  MoveL 6563 to (20.68, -72.48, -149.47) mm, rotated rx 105.8 ry 33.04 rz 34.05 deg; joints [-5.945, -30.892, 104.266, 145.331, 85.223, 18.714, -475]
  MoveL 6564 to (20.48, -73.16, -150.23) mm, rotated rx 105.8 ry 33.04 rz 34.05 deg; joints [-5.975, -30.911, 104.238, 145.3, 85.188, 18.748, -475]
  MoveL 6565 to (19.98, -73.73, -151.16) mm, rotated rx 105.8 ry 33.04 rz 34.05 deg; joints [-6.01, -30.911, 104.183, 145.262, 85.15, 18.787, -475]
  MoveL 6566 to (18.11, -74.59, -153.52) mm, rotated rx 105.8 ry 33.04 rz 34.05 deg; joints [-6.101, -30.851, 103.995, 145.167, 85.06, 18.882, -475]
  MoveL 6567 to (15.72, -74.84, -155.88) mm, rotated rx 105.8 ry 33.04 rz 34.05 deg; joints [-6.192, -30.738, 103.766, 145.073, 84.979, 18.97, -475]
  MoveL 6568 to (13.46, -74.3, -157.57) mm, rotated rx 105.8 ry 33.04 rz 34.05 deg; joints [-6.256, -30.597, 103.559, 145.006, 84.936, 19.024, -475]
  MoveL 6569 to (12.38, -73.73, -158.16) mm, rotated rx 105.8 ry 33.04 rz 34.05 deg; joints [-6.279, -30.516, 103.464, 144.984, 84.929, 19.037, -475]
  MoveL 6570 to (11.34, -72.97, -158.58) mm, rotated rx 105.8 ry 33.04 rz 34.05 deg; joints [-6.295, -30.429, 103.375, 144.968, 84.93, 19.042, -475]
  MoveL 6571 to (9.34, -70.84, -158.92) mm, rotated rx 105.8 ry 33.04 rz 34.05 deg; joints [-6.308, -30.233, 103.215, 144.957, 84.961, 19.025, -475]
  MoveL 6572 to (6.8, -67.51, -158.92) mm, rotated rx 105.8 ry 33.04 rz 34.05 deg; joints [-6.309, -29.957, 103.017, 144.96, 85.025, 18.98, -475]
  MoveL 6573 to (6.45, -67.09, -158.94) mm, rotated rx 105.8 ry 33.04 rz 34.05 deg; joints [-6.309, -29.921, 102.99, 144.96, 85.033, 18.975, -475]
  MoveL 6574 to (6.11, -66.68, -158.98) mm, rotated rx 105.8 ry 33.04 rz 34.05 deg; joints [-6.311, -29.886, 102.962, 144.959, 85.039, 18.971, -475]
  MoveL 6575 to (5.76, -66.29, -159.04) mm, rotated rx 105.8 ry 33.04 rz 34.05 deg; joints [-6.313, -29.85, 102.934, 144.957, 85.045, 18.968, -475]
  MoveL 6576 to (5.4, -65.92, -159.12) mm, rotated rx 105.8 ry 33.04 rz 34.05 deg; joints [-6.317, -29.815, 102.904, 144.954, 85.05, 18.965, -475]
  MoveL 6577 to (5.05, -65.55, -159.2) mm, rotated rx 105.8 ry 33.04 rz 34.05 deg; joints [-6.32, -29.781, 102.876, 144.951, 85.055, 18.963, -475]
  MoveL 6578 to (4.73, -65.18, -159.24) mm, rotated rx 105.8 ry 33.04 rz 34.05 deg; joints [-6.321, -29.749, 102.85, 144.95, 85.061, 18.959, -475]
  MoveL 6579 to (4.43, -64.8, -159.25) mm, rotated rx 105.8 ry 33.04 rz 34.05 deg; joints [-6.322, -29.717, 102.826, 144.95, 85.068, 18.955, -475]
  MoveL 6580 to (4.11, -64.39, -159.25) mm, rotated rx 105.8 ry 33.04 rz 34.05 deg; joints [-6.322, -29.683, 102.801, 144.95, 85.076, 18.949, -475]
  MoveL 6581 to (3.72, -63.9, -159.29) mm, rotated rx 105.8 ry 33.04 rz 34.05 deg; joints [-6.323, -29.641, 102.77, 144.949, 85.084, 18.944, -475]
  MoveL 6582 to (3.27, -63.39, -159.35) mm, rotated rx 105.8 ry 33.04 rz 34.05 deg; joints [-6.326, -29.596, 102.734, 144.947, 85.092, 18.939, -475]
  MoveL 6583 to (2.88, -62.94, -159.37) mm, rotated rx 105.8 ry 33.04 rz 34.05 deg; joints [-6.326, -29.556, 102.702, 144.947, 85.099, 18.934, -475]
  MoveL 6584 to (2.49, -62.55, -159.38) mm, rotated rx 105.8 ry 33.04 rz 34.05 deg; joints [-6.327, -29.518, 102.67, 144.947, 85.103, 18.932, -475]
  MoveL 6585 to (2.06, -62.19, -159.38) mm, rotated rx 105.8 ry 33.04 rz 34.05 deg; joints [-6.327, -29.481, 102.634, 144.947, 85.104, 18.931, -475]
  MoveL 6586 to (1.55, -61.92, -159.38) mm, rotated rx 105.8 ry 33.04 rz 34.05 deg; joints [-6.326, -29.443, 102.589, 144.947, 85.099, 18.935, -475]
  MoveL 6587 to (0.98, -61.7, -159.38) mm, rotated rx 105.8 ry 33.04 rz 34.05 deg; joints [-6.326, -29.404, 102.539, 144.947, 85.089, 18.941, -475]
  MoveL 6588 to (2.28, -62.59, -160.34) mm, rotated rx 105.8 ry 33.04 rz 34.05 deg; joints [-6.364, -29.51, 102.648, 144.91, 85.098, 18.948, -475]
  MoveL 6589 to (1.05, -62.41, -160.76) mm, rotated rx 105.8 ry 33.04 rz 34.05 deg; joints [-6.379, -29.438, 102.533, 144.893, 85.066, 18.977, -475]
  MoveL 6590 to (-0.34, -62.11, -161.09) mm, rotated rx 105.8 ry 33.04 rz 34.05 deg; joints [-6.391, -29.353, 102.406, 144.879, 85.033, 19.004, -475]
  MoveL 6591 to (-1.89, -61.69, -161.34) mm, rotated rx 105.8 ry 33.04 rz 34.05 deg; joints [-6.4, -29.255, 102.265, 144.869, 84.999, 19.031, -475]
  MoveL 6592 to (-3.92, -61.03, -161.45) mm, rotated rx 105.8 ry 33.04 rz 34.05 deg; joints [-6.402, -29.121, 102.081, 144.863, 84.959, 19.06, -475]
  MoveL 6593 to (-5.95, -60.38, -161.68) mm, rotated rx 105.8 ry 33.04 rz 34.05 deg; joints [-6.41, -28.988, 101.897, 144.854, 84.918, 19.091, -475]
  MoveL 6594 to (-7.97, -59.71, -161.79) mm, rotated rx 105.8 ry 33.04 rz 34.05 deg; joints [-6.413, -28.854, 101.713, 144.848, 84.878, 19.121, -475]
  MoveL 6595 to (-10, -59.04, -161.91) mm, rotated rx 105.8 ry 33.04 rz 34.05 deg; joints [-6.416, -28.72, 101.529, 144.843, 84.838, 19.151, -475]
  MoveL 6596 to (-12.02, -58.38, -162.14) mm, rotated rx 105.8 ry 33.04 rz 34.05 deg; joints [-6.424, -28.587, 101.344, 144.832, 84.797, 19.182, -475]
  MoveL 6597 to (-14.05, -57.7, -162.27) mm, rotated rx 105.8 ry 33.04 rz 34.05 deg; joints [-6.427, -28.453, 101.16, 144.827, 84.756, 19.212, -475]
  MoveL 6598 to (-16.07, -57.02, -162.38) mm, rotated rx 105.8 ry 33.04 rz 34.05 deg; joints [-6.43, -28.318, 100.975, 144.821, 84.716, 19.242, -475]
  MoveL 6599 to (-18.4, -56.24, -162.54) mm, rotated rx 105.8 ry 33.04 rz 34.05 deg; joints [-6.434, -28.164, 100.761, 144.813, 84.668, 19.277, -475]
  MoveL 6600 to (-20.39, -55.57, -162.74) mm, rotated rx 105.8 ry 33.04 rz 34.05 deg; joints [-6.44, -28.031, 100.579, 144.805, 84.628, 19.308, -475]
  MoveL 6601 to (-22.58, -54.83, -162.94) mm, rotated rx 105.8 ry 33.04 rz 34.05 deg; joints [-6.446, -27.885, 100.378, 144.796, 84.584, 19.342, -475]
  MoveL 6602 to (-24.71, -54.09, -163.19) mm, rotated rx 105.8 ry 33.04 rz 34.05 deg; joints [-6.454, -27.743, 100.18, 144.785, 84.541, 19.375, -475]
  MoveL 6603 to (-26.73, -53.4, -163.31) mm, rotated rx 105.8 ry 33.04 rz 34.05 deg; joints [-6.458, -27.608, 99.994, 144.779, 84.5, 19.406, -475]
  MoveL 6604 to (-28.75, -52.71, -163.31) mm, rotated rx 105.8 ry 33.04 rz 34.05 deg; joints [-6.456, -27.473, 99.808, 144.777, 84.457, 19.435, -475]
  MoveL 6605 to (-30.74, -52.02, -163.39) mm, rotated rx 105.8 ry 33.04 rz 34.05 deg; joints [-6.458, -27.34, 99.624, 144.773, 84.416, 19.465, -475]
  MoveL 6606 to (-32.68, -51.33, -163.6) mm, rotated rx 105.8 ry 33.04 rz 34.05 deg; joints [-6.465, -27.209, 99.444, 144.764, 84.377, 19.495, -475]
  MoveL 6607 to (-34.84, -50.54, -163.95) mm, rotated rx 105.8 ry 33.04 rz 34.05 deg; joints [-6.476, -27.062, 99.243, 144.749, 84.335, 19.53, -475]
  MoveL 6608 to (-36.54, -49.92, -164.16) mm, rotated rx 105.8 ry 33.04 rz 34.05 deg; joints [-6.483, -26.947, 99.085, 144.74, 84.301, 19.556, -475]
  MoveL 6609 to (-38.84, -49.05, -164.46) mm, rotated rx 105.8 ry 33.04 rz 34.05 deg; joints [-6.493, -26.79, 98.871, 144.727, 84.256, 19.592, -475]
  MoveL 6610 to (-40.92, -48.31, -164.57) mm, rotated rx 105.8 ry 33.04 rz 34.05 deg; joints [-6.496, -26.649, 98.676, 144.721, 84.213, 19.624, -475]
  MoveL 6611 to (-42.93, -47.62, -164.58) mm, rotated rx 105.8 ry 33.04 rz 34.05 deg; joints [-6.495, -26.515, 98.488, 144.719, 84.169, 19.655, -475]
  MoveL 6612 to (-43.47, -46.91, -165.37) mm, rotated rx 105.8 ry 33.04 rz 34.05 deg; joints [-6.525, -26.456, 98.44, 144.69, 84.183, 19.656, -475]
  MoveL 6613 to (-43.03, -46.88, -165.76) mm, rotated rx 105.8 ry 33.04 rz 34.05 deg; joints [-6.54, -26.477, 98.482, 144.677, 84.203, 19.648, -475]
  MoveL 6614 to (-42.89, -46.88, -166) mm, rotated rx 105.8 ry 33.04 rz 34.05 deg; joints [-6.55, -26.484, 98.495, 144.668, 84.209, 19.647, -475]
  MoveL 6615 to (-43.03, -46.91, -166.13) mm, rotated rx 105.8 ry 33.04 rz 34.05 deg; joints [-6.554, -26.479, 98.481, 144.663, 84.203, 19.653, -475]
  MoveL 6616 to (-43.41, -47, -166.15) mm, rotated rx 105.8 ry 33.04 rz 34.05 deg; joints [-6.554, -26.462, 98.442, 144.661, 84.185, 19.666, -475]
  MoveL 6617 to (-43.87, -47.11, -166.16) mm, rotated rx 105.8 ry 33.04 rz 34.05 deg; joints [-6.554, -26.443, 98.397, 144.66, 84.164, 19.681, -475]
  MoveL 6618 to (-45.38, -47.52, -166.16) mm, rotated rx 105.8 ry 33.04 rz 34.05 deg; joints [-6.552, -26.381, 98.246, 144.657, 84.091, 19.732, -475]
  MoveL 6619 to (-45.92, -47.65, -166.18) mm, rotated rx 105.8 ry 33.04 rz 34.05 deg; joints [-6.552, -26.358, 98.192, 144.655, 84.065, 19.75, -475]
  MoveL 6620 to (-46.46, -47.77, -166.22) mm, rotated rx 105.8 ry 33.04 rz 34.05 deg; joints [-6.553, -26.334, 98.138, 144.652, 84.041, 19.768, -475]
  MoveL 6621 to (-47.03, -47.86, -166.31) mm, rotated rx 105.8 ry 33.04 rz 34.05 deg; joints [-6.556, -26.309, 98.082, 144.648, 84.017, 19.786, -475]
  MoveL 6622 to (-47.57, -47.97, -166.37) mm, rotated rx 105.8 ry 33.04 rz 34.05 deg; joints [-6.557, -26.284, 98.028, 144.644, 83.992, 19.804, -475]
  MoveL 6623 to (-48.09, -48.09, -166.39) mm, rotated rx 105.8 ry 33.04 rz 34.05 deg; joints [-6.558, -26.262, 97.976, 144.642, 83.968, 19.821, -475]
  MoveL 6624 to (-48.57, -48.2, -166.41) mm, rotated rx 105.8 ry 33.04 rz 34.05 deg; joints [-6.558, -26.242, 97.928, 144.64, 83.946, 19.838, -475]
  MoveL 6625 to (-49.02, -48.29, -166.45) mm, rotated rx 105.8 ry 33.04 rz 34.05 deg; joints [-6.559, -26.222, 97.883, 144.638, 83.926, 19.852, -475]
  MoveL 6626 to (-49.45, -48.38, -166.49) mm, rotated rx 105.8 ry 33.04 rz 34.05 deg; joints [-6.56, -26.202, 97.839, 144.635, 83.906, 19.867, -475]
  MoveL 6627 to (-49.94, -48.5, -166.51) mm, rotated rx 105.8 ry 33.04 rz 34.05 deg; joints [-6.56, -26.182, 97.791, 144.634, 83.883, 19.883, -475]
  MoveL 6628 to (-50.51, -48.63, -166.53) mm, rotated rx 105.8 ry 33.04 rz 34.05 deg; joints [-6.56, -26.158, 97.734, 144.632, 83.857, 19.902, -475]
  MoveL 6629 to (-51.19, -48.77, -166.58) mm, rotated rx 105.8 ry 33.04 rz 34.05 deg; joints [-6.561, -26.127, 97.665, 144.628, 83.825, 19.925, -475]
  MoveL 6630 to (-51.78, -48.91, -166.61) mm, rotated rx 105.8 ry 33.04 rz 34.05 deg; joints [-6.561, -26.102, 97.606, 144.626, 83.798, 19.944, -475]
  MoveL 6631 to (-53.82, -49.45, -166.61) mm, rotated rx 105.8 ry 33.04 rz 34.05 deg; joints [-6.559, -26.017, 97.401, 144.62, 83.7, 20.014, -475]
  MoveL 6632 to (-56.69, -49.93, -166.94) mm, rotated rx 105.8 ry 33.04 rz 34.05 deg; joints [-6.568, -25.885, 97.113, 144.602, 83.575, 20.106, -475]
  MoveL 6633 to (-57.98, -49.9, -167.35) mm, rotated rx 105.8 ry 33.04 rz 34.05 deg; joints [-6.582, -25.815, 96.985, 144.584, 83.53, 20.144, -475]
  MoveL 6634 to (-59.18, -49.7, -167.93) mm, rotated rx 105.8 ry 33.04 rz 34.05 deg; joints [-6.602, -25.742, 96.867, 144.561, 83.497, 20.176, -475]
  MoveL 6635 to (-61.29, -48.77, -169.58) mm, rotated rx 105.8 ry 33.04 rz 34.05 deg; joints [-6.663, -25.59, 96.664, 144.498, 83.466, 20.222, -475]
  MoveL 6636 to (-63.02, -47.13, -171.89) mm, rotated rx 105.8 ry 33.04 rz 34.05 deg; joints [-6.749, -25.429, 96.502, 144.414, 83.482, 20.246, -475]
  MoveL 6637 to (-63.97, -45.34, -174.19) mm, rotated rx 105.8 ry 33.04 rz 34.05 deg; joints [-6.837, -25.302, 96.418, 144.331, 83.533, 20.244, -475]
  MoveL 6638 to (-64, -44.59, -175.1) mm, rotated rx 105.8 ry 33.04 rz 34.05 deg; joints [-6.872, -25.269, 96.418, 144.3, 83.567, 20.233, -475]
  MoveL 6639 to (-63.75, -43.94, -175.84) mm, rotated rx 105.8 ry 33.04 rz 34.05 deg; joints [-6.9, -25.255, 96.447, 144.274, 83.608, 20.215, -475]
  MoveL 6640 to (-63.51, -43.65, -176.15) mm, rotated rx 105.8 ry 33.04 rz 34.05 deg; joints [-6.913, -25.255, 96.472, 144.264, 83.63, 20.204, -475]
  MoveL 6641 to (-63.2, -43.39, -176.42) mm, rotated rx 105.8 ry 33.04 rz 34.05 deg; joints [-6.923, -25.26, 96.505, 144.255, 83.654, 20.191, -475]
  MoveL 6642 to (-62.36, -42.93, -176.83) mm, rotated rx 105.8 ry 33.04 rz 34.05 deg; joints [-6.94, -25.286, 96.591, 144.243, 83.707, 20.16, -475]
  MoveL 6643 to (-61.22, -42.58, -177.08) mm, rotated rx 105.8 ry 33.04 rz 34.05 deg; joints [-6.952, -25.33, 96.705, 144.236, 83.765, 20.122, -475]
  MoveL 6644 to (-59.79, -42.31, -177.16) mm, rotated rx 105.8 ry 33.04 rz 34.05 deg; joints [-6.957, -25.395, 96.848, 144.236, 83.83, 20.077, -475]
  MoveL 6645 to (-56.16, -41.83, -177.16) mm, rotated rx 105.8 ry 33.04 rz 34.05 deg; joints [-6.962, -25.566, 97.211, 144.243, 83.986, 19.966, -475]
  MoveL 6646 to (-55.7, -41.77, -177.14) mm, rotated rx 105.8 ry 33.04 rz 34.05 deg; joints [-6.962, -25.588, 97.256, 144.244, 84.005, 19.952, -475]
  MoveL 6647 to (-55.29, -41.74, -177.12) mm, rotated rx 105.8 ry 33.04 rz 34.05 deg; joints [-6.962, -25.608, 97.297, 144.246, 84.022, 19.94, -475]
  MoveL 6648 to (-54.82, -41.69, -177.1) mm, rotated rx 105.8 ry 33.04 rz 34.05 deg; joints [-6.962, -25.631, 97.344, 144.247, 84.041, 19.926, -475]
  MoveL 6649 to (-51.19, -41.2, -177.1) mm, rotated rx 105.8 ry 33.04 rz 34.05 deg; joints [-6.967, -25.801, 97.704, 144.254, 84.197, 19.815, -475]
  MoveL 6650 to (-50.65, -41.15, -177.08) mm, rotated rx 105.8 ry 33.04 rz 34.05 deg; joints [-6.967, -25.828, 97.758, 144.255, 84.218, 19.8, -475]
  MoveL 6651 to (-50.1, -41.13, -177.04) mm, rotated rx 105.8 ry 33.04 rz 34.05 deg; joints [-6.966, -25.855, 97.811, 144.257, 84.239, 19.784, -475]
  MoveL 6652 to (-49.62, -41.16, -177) mm, rotated rx 105.8 ry 33.04 rz 34.05 deg; joints [-6.965, -25.882, 97.859, 144.26, 84.256, 19.772, -475]
  MoveL 6653 to (-49.24, -41.22, -176.94) mm, rotated rx 105.8 ry 33.04 rz 34.05 deg; joints [-6.963, -25.905, 97.895, 144.262, 84.267, 19.763, -475]
  MoveL 6654 to (-49.06, -41.28, -176.77) mm, rotated rx 105.8 ry 33.04 rz 34.05 deg; joints [-6.957, -25.917, 97.913, 144.269, 84.27, 19.758, -475]
  MoveL 6655 to (-49.05, -41.32, -176.44) mm, rotated rx 105.8 ry 33.04 rz 34.05 deg; joints [-6.945, -25.919, 97.915, 144.281, 84.268, 19.755, -475]
  MoveL 6656 to (-49.2, -41.32, -175.93) mm, rotated rx 105.8 ry 33.04 rz 34.05 deg; joints [-6.925, -25.912, 97.901, 144.3, 84.26, 19.754, -475]
  MoveL 6657 to (-48.89, -42.09, -174.47) mm, rotated rx 105.8 ry 33.04 rz 34.05 deg; joints [-6.869, -25.962, 97.929, 144.353, 84.232, 19.753, -475]
  MoveL 6658 to (-45.07, -43.97, -174.47) mm, rotated rx 105.8 ry 33.04 rz 34.05 deg; joints [-6.872, -26.242, 98.284, 144.354, 84.293, 19.71, -475]
  MoveL 6659 to (-43.24, -44.88, -174.42) mm, rotated rx 105.8 ry 33.04 rz 34.05 deg; joints [-6.872, -26.376, 98.453, 144.357, 84.321, 19.689, -475]
  MoveL 6660 to (-41.47, -45.76, -174.33) mm, rotated rx 105.8 ry 33.04 rz 34.05 deg; joints [-6.87, -26.506, 98.617, 144.361, 84.348, 19.669, -475]
  MoveL 6661 to (-39.66, -46.65, -174.25) mm, rotated rx 105.8 ry 33.04 rz 34.05 deg; joints [-6.868, -26.639, 98.784, 144.364, 84.375, 19.649, -475]
  MoveL 6662 to (-37.89, -47.52, -174.15) mm, rotated rx 105.8 ry 33.04 rz 34.05 deg; joints [-6.866, -26.769, 98.946, 144.369, 84.401, 19.629, -475]
  MoveL 6663 to (-36.03, -48.47, -174.11) mm, rotated rx 105.8 ry 33.04 rz 34.05 deg; joints [-6.866, -26.907, 99.117, 144.371, 84.428, 19.61, -475]
  MoveL 6664 to (-34.1, -49.54, -174.07) mm, rotated rx 105.8 ry 33.04 rz 34.05 deg; joints [-6.866, -27.053, 99.292, 144.372, 84.452, 19.593, -475]
  MoveL 6665 to (-31.82, -50.56, -173.91) mm, rotated rx 105.8 ry 33.04 rz 34.05 deg; joints [-6.861, -27.215, 99.502, 144.379, 84.489, 19.564, -475]
  MoveL 6666 to (-29.81, -51.55, -173.66) mm, rotated rx 105.8 ry 33.04 rz 34.05 deg; joints [-6.853, -27.363, 99.686, 144.389, 84.518, 19.54, -475]
  MoveL 6667 to (-27.84, -52.52, -173.53) mm, rotated rx 105.8 ry 33.04 rz 34.05 deg; joints [-6.85, -27.507, 99.866, 144.394, 84.546, 19.519, -475]
  MoveL 6668 to (-25.92, -53.46, -173.29) mm, rotated rx 105.8 ry 33.04 rz 34.05 deg; joints [-6.842, -27.647, 100.04, 144.404, 84.573, 19.497, -475]
  MoveL 6669 to (-24, -54.39, -173.17) mm, rotated rx 105.8 ry 33.04 rz 34.05 deg; joints [-6.839, -27.787, 100.214, 144.409, 84.6, 19.476, -475]
  MoveL 6670 to (-22.08, -55.33, -173.05) mm, rotated rx 105.8 ry 33.04 rz 34.05 deg; joints [-6.836, -27.927, 100.388, 144.414, 84.626, 19.456, -475]
  MoveL 6671 to (-20.16, -56.25, -172.81) mm, rotated rx 105.8 ry 33.04 rz 34.05 deg; joints [-6.828, -28.067, 100.562, 144.423, 84.653, 19.434, -475]
  MoveL 6672 to (-18.24, -57.18, -172.69) mm, rotated rx 105.8 ry 33.04 rz 34.05 deg; joints [-6.825, -28.207, 100.736, 144.428, 84.68, 19.413, -475]
  MoveL 6673 to (-16.32, -58.1, -172.57) mm, rotated rx 105.8 ry 33.04 rz 34.05 deg; joints [-6.822, -28.347, 100.909, 144.432, 84.707, 19.393, -475]
  MoveL 6674 to (-14.39, -59.03, -172.45) mm, rotated rx 105.8 ry 33.04 rz 34.05 deg; joints [-6.819, -28.486, 101.081, 144.437, 84.733, 19.373, -475]
  MoveL 6675 to (-12.46, -59.93, -172.22) mm, rotated rx 105.8 ry 33.04 rz 34.05 deg; joints [-6.812, -28.626, 101.255, 144.446, 84.76, 19.351, -475]
  MoveL 6676 to (-10.53, -60.85, -172.11) mm, rotated rx 105.8 ry 33.04 rz 34.05 deg; joints [-6.809, -28.765, 101.428, 144.451, 84.786, 19.331, -475]
  MoveL 6677 to (-8.9, -61.58, -171.86) mm, rotated rx 105.8 ry 33.04 rz 34.05 deg; joints [-6.801, -28.882, 101.574, 144.46, 84.809, 19.312, -475]
  MoveL 6678 to (-7.39, -62.24, -171.54) mm, rotated rx 105.8 ry 33.04 rz 34.05 deg; joints [-6.789, -28.989, 101.711, 144.473, 84.831, 19.292, -475]
  MoveL 6679 to (-5.94, -62.84, -171.12) mm, rotated rx 105.8 ry 33.04 rz 34.05 deg; joints [-6.774, -29.09, 101.843, 144.489, 84.853, 19.271, -475]
  MoveL 6680 to (-7.04, -61.5, -170.16) mm, rotated rx 105.8 ry 33.04 rz 34.05 deg; joints [-6.737, -28.976, 101.756, 144.527, 84.87, 19.245, -475]
  MoveL 6681 to (-6.5, -61.82, -170.04) mm, rotated rx 105.8 ry 33.04 rz 34.05 deg; joints [-6.733, -29.018, 101.805, 144.532, 84.874, 19.24, -475]
  MoveL 6682 to (-6.03, -62.17, -169.95) mm, rotated rx 105.8 ry 33.04 rz 34.05 deg; joints [-6.729, -29.057, 101.845, 144.535, 84.874, 19.239, -475]
  MoveL 6683 to (-5.66, -62.57, -169.92) mm, rotated rx 105.8 ry 33.04 rz 34.05 deg; joints [-6.728, -29.093, 101.875, 144.536, 84.869, 19.242, -475]
  MoveL 6684 to (-5.35, -63, -169.9) mm, rotated rx 105.8 ry 33.04 rz 34.05 deg; joints [-6.728, -29.128, 101.9, 144.536, 84.861, 19.248, -475]
  MoveL 6685 to (-3.48, -66.17, -169.89) mm, rotated rx 105.8 ry 33.04 rz 34.05 deg; joints [-6.726, -29.361, 102.039, 144.532, 84.784, 19.302, -475]
  MoveL 6686 to (-3.24, -66.57, -169.88) mm, rotated rx 105.8 ry 33.04 rz 34.05 deg; joints [-6.726, -29.391, 102.057, 144.532, 84.775, 19.309, -475]
  MoveL 6687 to (-3.02, -66.92, -169.85) mm, rotated rx 105.8 ry 33.04 rz 34.05 deg; joints [-6.725, -29.418, 102.075, 144.533, 84.766, 19.314, -475]
  MoveL 6688 to (-2.77, -67.33, -169.84) mm, rotated rx 105.8 ry 33.04 rz 34.05 deg; joints [-6.724, -29.449, 102.093, 144.532, 84.756, 19.321, -475]
  MoveL 6689 to (-2.51, -67.79, -169.84) mm, rotated rx 105.8 ry 33.04 rz 34.05 deg; joints [-6.724, -29.482, 102.113, 144.532, 84.745, 19.329, -475]
  MoveL 6690 to (-1.72, -69.15, -169.84) mm, rotated rx 105.8 ry 33.04 rz 34.05 deg; joints [-6.724, -29.581, 102.17, 144.53, 84.711, 19.353, -475]
  MoveL 6691 to (-1.4, -69.68, -169.82) mm, rotated rx 105.8 ry 33.04 rz 34.05 deg; joints [-6.723, -29.621, 102.195, 144.53, 84.699, 19.362, -475]
  MoveL 6692 to (-1.01, -70.29, -169.78) mm, rotated rx 105.8 ry 33.04 rz 34.05 deg; joints [-6.721, -29.667, 102.224, 144.531, 84.684, 19.372, -475]
  MoveL 6693 to (-0.68, -70.84, -169.76) mm, rotated rx 105.8 ry 33.04 rz 34.05 deg; joints [-6.72, -29.708, 102.249, 144.531, 84.671, 19.381, -475]
  MoveL 6694 to (-0.15, -71.75, -169.76) mm, rotated rx 105.8 ry 33.04 rz 34.05 deg; joints [-6.72, -29.774, 102.287, 144.529, 84.648, 19.397, -475]
  MoveL 6695 to (0.51, -73.03, -169.85) mm, rotated rx 105.8 ry 33.04 rz 34.05 deg; joints [-6.723, -29.864, 102.333, 144.524, 84.614, 19.423, -475]
  MoveL 6696 to (0.91, -74.15, -170.1) mm, rotated rx 105.8 ry 33.04 rz 34.05 deg; joints [-6.732, -29.933, 102.357, 144.513, 84.579, 19.452, -475]
  MoveL 6697 to (1.06, -75.09, -170.52) mm, rotated rx 105.8 ry 33.04 rz 34.05 deg; joints [-6.748, -29.98, 102.358, 144.495, 84.543, 19.483, -475]
  MoveL 6698 to (1.03, -75.5, -170.79) mm, rotated rx 105.8 ry 33.04 rz 34.05 deg; joints [-6.758, -29.996, 102.35, 144.484, 84.525, 19.499, -475]
  MoveL 6699 to (0.94, -75.86, -171.11) mm, rotated rx 105.8 ry 33.04 rz 34.05 deg; joints [-6.77, -30.007, 102.336, 144.471, 84.507, 19.517, -475]
  MoveL 6700 to (0.57, -76.45, -171.86) mm, rotated rx 105.8 ry 33.04 rz 34.05 deg; joints [-6.798, -30.012, 102.291, 144.44, 84.472, 19.553, -475]
  MoveL 6701 to (-0.07, -76.88, -172.79) mm, rotated rx 105.8 ry 33.04 rz 34.05 deg; joints [-6.833, -29.997, 102.223, 144.404, 84.435, 19.592, -475]
  MoveL 6702 to (-2.11, -77.2, -175.14) mm, rotated rx 105.8 ry 33.04 rz 34.05 deg; joints [-6.921, -29.902, 102.019, 144.311, 84.363, 19.678, -475]
  MoveL 6703 to (-4.51, -76.81, -177.49) mm, rotated rx 105.8 ry 33.04 rz 34.05 deg; joints [-7.009, -29.758, 101.79, 144.22, 84.309, 19.75, -475]
  MoveL 6704 to (-6.57, -75.7, -179.17) mm, rotated rx 105.8 ry 33.04 rz 34.05 deg; joints [-7.073, -29.601, 101.604, 144.157, 84.296, 19.784, -475]
  MoveL 6705 to (-7.48, -74.87, -179.76) mm, rotated rx 105.8 ry 33.04 rz 34.05 deg; joints [-7.095, -29.518, 101.526, 144.135, 84.305, 19.786, -475]
  MoveL 6706 to (-8.3, -73.86, -180.18) mm, rotated rx 105.8 ry 33.04 rz 34.05 deg; joints [-7.111, -29.432, 101.46, 144.12, 84.324, 19.778, -475]
  MoveL 6707 to (-9.69, -71.29, -180.51) mm, rotated rx 105.8 ry 33.04 rz 34.05 deg; joints [-7.125, -29.25, 101.358, 144.112, 84.391, 19.734, -475]
  MoveL 6708 to (-10.89, -68.39, -180.51) mm, rotated rx 105.8 ry 33.04 rz 34.05 deg; joints [-7.126, -29.063, 101.278, 144.117, 84.478, 19.672, -475]
  MoveL 6709 to (-11.32, -67.51, -180.56) mm, rotated rx 105.8 ry 33.04 rz 34.05 deg; joints [-7.128, -29.004, 101.248, 144.116, 84.503, 19.655, -475]
  MoveL 6710 to (-11.52, -67.02, -180.56) mm, rotated rx 105.8 ry 33.04 rz 34.05 deg; joints [-7.128, -28.972, 101.235, 144.117, 84.517, 19.644, -475]
  MoveL 6711 to (-11.73, -66.52, -180.56) mm, rotated rx 105.8 ry 33.04 rz 34.05 deg; joints [-7.129, -28.94, 101.221, 144.118, 84.532, 19.634, -475]
  MoveL 6712 to (-11.96, -66.01, -180.59) mm, rotated rx 105.8 ry 33.04 rz 34.05 deg; joints [-7.13, -28.906, 101.205, 144.118, 84.547, 19.623, -475]
  MoveL 6713 to (-12.24, -65.42, -180.65) mm, rotated rx 105.8 ry 33.04 rz 34.05 deg; joints [-7.132, -28.866, 101.184, 144.116, 84.563, 19.613, -475]
  MoveL 6714 to (-12.48, -64.9, -180.68) mm, rotated rx 105.8 ry 33.04 rz 34.05 deg; joints [-7.134, -28.831, 101.167, 144.116, 84.578, 19.602, -475]
  MoveL 6715 to (-12.69, -64.42, -180.69) mm, rotated rx 105.8 ry 33.04 rz 34.05 deg; joints [-7.134, -28.8, 101.153, 144.116, 84.592, 19.593, -475]
  MoveL 6716 to (-12.9, -63.98, -180.72) mm, rotated rx 105.8 ry 33.04 rz 34.05 deg; joints [-7.136, -28.771, 101.138, 144.116, 84.604, 19.584, -475]
  MoveL 6717 to (-13.1, -63.58, -180.77) mm, rotated rx 105.8 ry 33.04 rz 34.05 deg; joints [-7.138, -28.743, 101.123, 144.114, 84.615, 19.577, -475]
  MoveL 6718 to (-13.31, -63.17, -180.81) mm, rotated rx 105.8 ry 33.04 rz 34.05 deg; joints [-7.139, -28.714, 101.108, 144.114, 84.626, 19.57, -475]
  MoveL 6719 to (-13.51, -62.7, -180.82) mm, rotated rx 105.8 ry 33.04 rz 34.05 deg; joints [-7.14, -28.684, 101.094, 144.114, 84.639, 19.56, -475]
  MoveL 6720 to (-13.72, -62.23, -180.83) mm, rotated rx 105.8 ry 33.04 rz 34.05 deg; joints [-7.14, -28.653, 101.079, 144.114, 84.652, 19.551, -475]
  MoveL 6721 to (-13.95, -61.77, -180.83) mm, rotated rx 105.8 ry 33.04 rz 34.05 deg; joints [-7.141, -28.621, 101.063, 144.115, 84.665, 19.542, -475]
  MoveL 6722 to (-14.22, -61.36, -180.85) mm, rotated rx 105.8 ry 33.04 rz 34.05 deg; joints [-7.142, -28.589, 101.042, 144.115, 84.674, 19.536, -475]
  MoveL 6723 to (-14.52, -60.99, -180.88) mm, rotated rx 105.8 ry 33.04 rz 34.05 deg; joints [-7.143, -28.558, 101.017, 144.114, 84.679, 19.532, -475]
  MoveL 6724 to (-14.86, -60.69, -180.93) mm, rotated rx 105.8 ry 33.04 rz 34.05 deg; joints [-7.144, -28.527, 100.988, 144.112, 84.681, 19.532, -475]
  MoveL 6725 to (-15.22, -60.41, -180.97) mm, rotated rx 105.8 ry 33.04 rz 34.05 deg; joints [-7.146, -28.496, 100.957, 144.111, 84.681, 19.532, -475]
  MoveL 6726 to (-14.19, -61.53, -181.94) mm, rotated rx 105.8 ry 33.04 rz 34.05 deg; joints [-7.183, -28.597, 101.038, 144.073, 84.672, 19.553, -475]
  MoveL 6727 to (-15.71, -60.73, -182.32) mm, rotated rx 105.8 ry 33.04 rz 34.05 deg; joints [-7.197, -28.483, 100.901, 144.059, 84.655, 19.57, -475]
  MoveL 6728 to (-17.29, -59.83, -182.6) mm, rotated rx 105.8 ry 33.04 rz 34.05 deg; joints [-7.206, -28.363, 100.761, 144.049, 84.641, 19.584, -475]
  MoveL 6729 to (-18.95, -58.82, -182.8) mm, rotated rx 105.8 ry 33.04 rz 34.05 deg; joints [-7.212, -28.233, 100.613, 144.042, 84.628, 19.596, -475]
  MoveL 6730 to (-20.76, -57.68, -183.02) mm, rotated rx 105.8 ry 33.04 rz 34.05 deg; joints [-7.219, -28.09, 100.452, 144.034, 84.615, 19.608, -475]
  MoveL 6731 to (-22.55, -56.52, -183.14) mm, rotated rx 105.8 ry 33.04 rz 34.05 deg; joints [-7.222, -27.947, 100.294, 144.03, 84.602, 19.618, -475]
  MoveL 6732 to (-24.34, -55.36, -183.25) mm, rotated rx 105.8 ry 33.04 rz 34.05 deg; joints [-7.225, -27.804, 100.135, 144.026, 84.59, 19.628, -475]
  MoveL 6733 to (-26.14, -54.21, -183.48) mm, rotated rx 105.8 ry 33.04 rz 34.05 deg; joints [-7.233, -27.66, 99.974, 144.018, 84.577, 19.64, -475]
  MoveL 6734 to (-27.92, -53.04, -183.6) mm, rotated rx 105.8 ry 33.04 rz 34.05 deg; joints [-7.236, -27.517, 99.814, 144.014, 84.565, 19.651, -475]
  MoveL 6735 to (-29.71, -51.87, -183.72) mm, rotated rx 105.8 ry 33.04 rz 34.05 deg; joints [-7.239, -27.374, 99.655, 144.01, 84.552, 19.661, -475]
  MoveL 6736 to (-31.5, -50.7, -183.96) mm, rotated rx 105.8 ry 33.04 rz 34.05 deg; joints [-7.247, -27.231, 99.494, 144.002, 84.539, 19.673, -475]
  MoveL 6737 to (-33.28, -49.53, -184.08) mm, rotated rx 105.8 ry 33.04 rz 34.05 deg; joints [-7.25, -27.088, 99.334, 143.998, 84.526, 19.684, -475]
  MoveL 6738 to (-35.06, -48.35, -184.2) mm, rotated rx 105.8 ry 33.04 rz 34.05 deg; joints [-7.253, -26.944, 99.174, 143.994, 84.513, 19.695, -475]
  MoveL 6739 to (-36.74, -47.23, -184.39) mm, rotated rx 105.8 ry 33.04 rz 34.05 deg; joints [-7.259, -26.809, 99.022, 143.987, 84.501, 19.706, -475]
  MoveL 6740 to (-38.26, -46.22, -184.6) mm, rotated rx 105.8 ry 33.04 rz 34.05 deg; joints [-7.266, -26.686, 98.884, 143.979, 84.49, 19.716, -475]
  MoveL 6741 to (-39.89, -45.13, -184.71) mm, rotated rx 105.8 ry 33.04 rz 34.05 deg; joints [-7.269, -26.554, 98.737, 143.976, 84.478, 19.727, -475]
  MoveL 6742 to (-41.75, -44.01, -184.71) mm, rotated rx 105.8 ry 33.04 rz 34.05 deg; joints [-7.267, -26.409, 98.567, 143.976, 84.457, 19.741, -475]
  MoveL 6743 to (-44.01, -42.49, -184.8) mm, rotated rx 105.8 ry 33.04 rz 34.05 deg; joints [-7.269, -26.226, 98.362, 143.973, 84.44, 19.754, -475]
  MoveL 6744 to (-45.98, -41.02, -185.04) mm, rotated rx 105.8 ry 33.04 rz 34.05 deg; joints [-7.276, -26.06, 98.183, 143.965, 84.43, 19.764, -475]
  MoveL 6745 to (-47.67, -39.88, -185.22) mm, rotated rx 105.8 ry 33.04 rz 34.05 deg; joints [-7.282, -25.923, 98.029, 143.958, 84.418, 19.775, -475]
  MoveL 6746 to (-49.2, -38.81, -185.54) mm, rotated rx 105.8 ry 33.04 rz 34.05 deg; joints [-7.293, -25.797, 97.887, 143.947, 84.407, 19.787, -475]
  MoveL 6747 to (-50.89, -37.65, -185.72) mm, rotated rx 105.8 ry 33.04 rz 34.05 deg; joints [-7.298, -25.66, 97.732, 143.94, 84.394, 19.799, -475]
  MoveL 6748 to (-52.51, -36.52, -185.92) mm, rotated rx 105.8 ry 33.04 rz 34.05 deg; joints [-7.305, -25.527, 97.584, 143.933, 84.383, 19.81, -475]
  MoveL 6749 to (-54.07, -35.4, -186.2) mm, rotated rx 105.8 ry 33.04 rz 34.05 deg; joints [-7.314, -25.397, 97.439, 143.923, 84.373, 19.82, -475]
  MoveL 6750 to (-54.37, -34.54, -186.97) mm, rotated rx 105.8 ry 33.04 rz 34.05 deg; joints [-7.344, -25.344, 97.414, 143.896, 84.401, 19.811, -475]
  MoveL 6751 to (-54, -34.56, -187.35) mm, rotated rx 105.8 ry 33.04 rz 34.05 deg; joints [-7.359, -25.364, 97.449, 143.882, 84.415, 19.807, -475]
  MoveL 6752 to (-53.92, -34.54, -187.59) mm, rotated rx 105.8 ry 33.04 rz 34.05 deg; joints [-7.368, -25.367, 97.456, 143.873, 84.42, 19.806, -475]
  MoveL 6753 to (-54.12, -34.48, -187.72) mm, rotated rx 105.8 ry 33.04 rz 34.05 deg; joints [-7.373, -25.354, 97.436, 143.868, 84.415, 19.812, -475]
  MoveL 6754 to (-54.65, -34.43, -187.77) mm, rotated rx 105.8 ry 33.04 rz 34.05 deg; joints [-7.374, -25.324, 97.385, 143.866, 84.399, 19.824, -475]
  MoveL 6755 to (-55.31, -34.38, -187.81) mm, rotated rx 105.8 ry 33.04 rz 34.05 deg; joints [-7.374, -25.287, 97.32, 143.864, 84.376, 19.841, -475]
  MoveL 6756 to (-56.88, -34.39, -187.81) mm, rotated rx 105.8 ry 33.04 rz 34.05 deg; joints [-7.372, -25.205, 97.165, 143.862, 84.317, 19.884, -475]
  MoveL 6757 to (-57.43, -34.39, -187.81) mm, rotated rx 105.8 ry 33.04 rz 34.05 deg; joints [-7.371, -25.176, 97.111, 143.861, 84.297, 19.898, -475]
  MoveL 6758 to (-57.97, -34.37, -187.84) mm, rotated rx 105.8 ry 33.04 rz 34.05 deg; joints [-7.371, -25.147, 97.059, 143.86, 84.277, 19.913, -475]
  MoveL 6759 to (-58.52, -34.34, -187.89) mm, rotated rx 105.8 ry 33.04 rz 34.05 deg; joints [-7.372, -25.117, 97.005, 143.857, 84.258, 19.927, -475]
  MoveL 6760 to (-59.07, -34.29, -187.96) mm, rotated rx 105.8 ry 33.04 rz 34.05 deg; joints [-7.374, -25.086, 96.95, 143.854, 84.24, 19.941, -475]
  MoveL 6761 to (-59.62, -34.25, -188.02) mm, rotated rx 105.8 ry 33.04 rz 34.05 deg; joints [-7.376, -25.055, 96.896, 143.851, 84.221, 19.955, -475]
  MoveL 6762 to (-60.12, -34.24, -188.04) mm, rotated rx 105.8 ry 33.04 rz 34.05 deg; joints [-7.376, -25.028, 96.847, 143.85, 84.203, 19.969, -475]
  MoveL 6763 to (-60.58, -34.23, -188.06) mm, rotated rx 105.8 ry 33.04 rz 34.05 deg; joints [-7.376, -25.004, 96.802, 143.849, 84.186, 19.981, -475]
  MoveL 6764 to (-62.15, -34.24, -188.06) mm, rotated rx 105.8 ry 33.04 rz 34.05 deg; joints [-7.373, -24.922, 96.647, 143.847, 84.127, 20.023, -475]
  MoveL 6765 to (-62.67, -34.23, -188.07) mm, rotated rx 105.8 ry 33.04 rz 34.05 deg; joints [-7.373, -24.894, 96.595, 143.845, 84.108, 20.037, -475]
  MoveL 6766 to (-63.14, -34.21, -188.1) mm, rotated rx 105.8 ry 33.04 rz 34.05 deg; joints [-7.373, -24.868, 96.548, 143.844, 84.091, 20.05, -475]
  MoveL 6767 to (-63.59, -34.18, -188.15) mm, rotated rx 105.8 ry 33.04 rz 34.05 deg; joints [-7.375, -24.843, 96.505, 143.842, 84.076, 20.061, -475]
  MoveL 6768 to (-64.04, -34.15, -188.19) mm, rotated rx 105.8 ry 33.04 rz 34.05 deg; joints [-7.375, -24.818, 96.46, 143.84, 84.06, 20.073, -475]
  MoveL 6769 to (-64.53, -34.14, -188.2) mm, rotated rx 105.8 ry 33.04 rz 34.05 deg; joints [-7.375, -24.792, 96.411, 143.838, 84.042, 20.087, -475]
  MoveL 6770 to (-65.05, -34.15, -188.2) mm, rotated rx 105.8 ry 33.04 rz 34.05 deg; joints [-7.374, -24.764, 96.359, 143.838, 84.022, 20.101, -475]
  MoveL 6771 to (-67.97, -33.87, -188.54) mm, rotated rx 105.8 ry 33.04 rz 34.05 deg; joints [-7.383, -24.598, 96.071, 143.822, 83.926, 20.175, -475]
  MoveL 6772 to (-69.23, -33.5, -188.96) mm, rotated rx 105.8 ry 33.04 rz 34.05 deg; joints [-7.397, -24.515, 95.947, 143.805, 83.894, 20.204, -475]
  MoveL 6773 to (-70.37, -33, -189.55) mm, rotated rx 105.8 ry 33.04 rz 34.05 deg; joints [-7.418, -24.433, 95.836, 143.783, 83.875, 20.227, -475]
  MoveL 6774 to (-72.26, -31.53, -191.24) mm, rotated rx 105.8 ry 33.04 rz 34.05 deg; joints [-7.48, -24.27, 95.653, 143.721, 83.871, 20.254, -475]
  MoveL 6775 to (-73.62, -29.48, -193.6) mm, rotated rx 105.8 ry 33.04 rz 34.05 deg; joints [-7.569, -24.109, 95.523, 143.637, 83.913, 20.259, -475]
  MoveL 6776 to (-74.2, -27.48, -195.96) mm, rotated rx 105.8 ry 33.04 rz 34.05 deg; joints [-7.659, -23.992, 95.471, 143.553, 83.982, 20.243, -475]
  MoveL 6777 to (-74.09, -26.73, -196.89) mm, rotated rx 105.8 ry 33.04 rz 34.05 deg; joints [-7.694, -23.965, 95.484, 143.521, 84.021, 20.229, -475]
  MoveL 6778 to (-73.71, -26.16, -197.65) mm, rotated rx 105.8 ry 33.04 rz 34.05 deg; joints [-7.724, -23.96, 95.522, 143.494, 84.061, 20.21, -475]
  MoveL 6779 to (-73.43, -25.94, -197.97) mm, rotated rx 105.8 ry 33.04 rz 34.05 deg; joints [-7.737, -23.966, 95.551, 143.483, 84.083, 20.199, -475]
  MoveL 6780 to (-73.07, -25.76, -198.24) mm, rotated rx 105.8 ry 33.04 rz 34.05 deg; joints [-7.748, -23.976, 95.587, 143.474, 84.105, 20.187, -475]
  MoveL 6781 to (-72.16, -25.53, -198.66) mm, rotated rx 105.8 ry 33.04 rz 34.05 deg; joints [-7.766, -24.014, 95.677, 143.46, 84.15, 20.16, -475]
  MoveL 6782 to (-70.98, -25.47, -198.92) mm, rotated rx 105.8 ry 33.04 rz 34.05 deg; joints [-7.778, -24.073, 95.794, 143.452, 84.199, 20.129, -475]
  MoveL 6783 to (-69.54, -25.58, -199) mm, rotated rx 105.8 ry 33.04 rz 34.05 deg; joints [-7.783, -24.154, 95.936, 143.45, 84.249, 20.093, -475]
  MoveL 6784 to (-67.98, -25.77, -199) mm, rotated rx 105.8 ry 33.04 rz 34.05 deg; joints [-7.786, -24.244, 96.089, 143.451, 84.3, 20.056, -475]
  MoveL 6785 to (-67.46, -25.84, -199) mm, rotated rx 105.8 ry 33.04 rz 34.05 deg; joints [-7.786, -24.275, 96.141, 143.452, 84.317, 20.044, -475]
  MoveL 6786 to (-66.89, -25.93, -198.96) mm, rotated rx 105.8 ry 33.04 rz 34.05 deg; joints [-7.786, -24.309, 96.197, 143.454, 84.335, 20.031, -475]
  MoveL 6787 to (-66.26, -26.06, -198.9) mm, rotated rx 105.8 ry 33.04 rz 34.05 deg; joints [-7.785, -24.347, 96.259, 143.456, 84.353, 20.016, -475]
  MoveL 6788 to (-65.7, -26.15, -198.87) mm, rotated rx 105.8 ry 33.04 rz 34.05 deg; joints [-7.785, -24.38, 96.313, 143.458, 84.371, 20.004, -475]
  MoveL 6789 to (-65.18, -26.22, -198.87) mm, rotated rx 105.8 ry 33.04 rz 34.05 deg; joints [-7.785, -24.411, 96.365, 143.458, 84.388, 19.991, -475]
  MoveL 6790 to (-64.66, -26.29, -198.86) mm, rotated rx 105.8 ry 33.04 rz 34.05 deg; joints [-7.786, -24.441, 96.415, 143.459, 84.404, 19.979, -475]
  MoveL 6791 to (-64.16, -26.38, -198.81) mm, rotated rx 105.8 ry 33.04 rz 34.05 deg; joints [-7.785, -24.471, 96.464, 143.461, 84.419, 19.968, -475]
  MoveL 6792 to (-63.67, -26.5, -198.73) mm, rotated rx 105.8 ry 33.04 rz 34.05 deg; joints [-7.783, -24.502, 96.512, 143.464, 84.432, 19.957, -475]
  MoveL 6793 to (-63.18, -26.63, -198.64) mm, rotated rx 105.8 ry 33.04 rz 34.05 deg; joints [-7.78, -24.533, 96.56, 143.468, 84.445, 19.946, -475]
  MoveL 6794 to (-62.68, -26.74, -198.57) mm, rotated rx 105.8 ry 33.04 rz 34.05 deg; joints [-7.778, -24.564, 96.609, 143.471, 84.459, 19.935, -475]
  MoveL 6795 to (-62.16, -26.82, -198.54) mm, rotated rx 105.8 ry 33.04 rz 34.05 deg; joints [-7.778, -24.595, 96.66, 143.472, 84.475, 19.923, -475]
  MoveL 6796 to (-61.65, -26.89, -198.53) mm, rotated rx 105.8 ry 33.04 rz 34.05 deg; joints [-7.778, -24.625, 96.71, 143.473, 84.492, 19.911, -475]
  MoveL 6797 to (-59.11, -27.25, -198.52) mm, rotated rx 105.8 ry 33.04 rz 34.05 deg; joints [-7.782, -24.773, 96.957, 143.475, 84.572, 19.853, -475]
  MoveL 6798 to (-58.74, -27.36, -198.5) mm, rotated rx 105.8 ry 33.04 rz 34.05 deg; joints [-7.782, -24.797, 96.993, 143.476, 84.581, 19.845, -475]
  MoveL 6799 to (-58.59, -27.43, -198.38) mm, rotated rx 105.8 ry 33.04 rz 34.05 deg; joints [-7.777, -24.808, 97.008, 143.48, 84.584, 19.842, -475]
  MoveL 6800 to (-58.68, -27.41, -198.15) mm, rotated rx 105.8 ry 33.04 rz 34.05 deg; joints [-7.769, -24.803, 97.001, 143.489, 84.581, 19.841, -475]
  MoveL 6801 to (-59.01, -27.27, -197.79) mm, rotated rx 105.8 ry 33.04 rz 34.05 deg; joints [-7.754, -24.78, 96.971, 143.502, 84.572, 19.842, -475]
  MoveL 6802 to (-58.8, -28.01, -197.05) mm, rotated rx 105.8 ry 33.04 rz 34.05 deg; joints [-7.726, -24.824, 96.989, 143.528, 84.547, 19.85, -475]
  MoveL 6803 to (-57.2, -29.4, -197.03) mm, rotated rx 105.8 ry 33.04 rz 34.05 deg; joints [-7.726, -24.967, 97.135, 143.528, 84.549, 19.848, -475]
  MoveL 6804 to (-55.57, -30.86, -196.9) mm, rotated rx 105.8 ry 33.04 rz 34.05 deg; joints [-7.723, -25.114, 97.283, 143.532, 84.549, 19.847, -475]
  MoveL 6805 to (-53.9, -32.4, -196.64) mm, rotated rx 105.8 ry 33.04 rz 34.05 deg; joints [-7.714, -25.268, 97.435, 143.54, 84.546, 19.846, -475]
  MoveL 6806 to (-52.32, -33.82, -196.51) mm, rotated rx 105.8 ry 33.04 rz 34.05 deg; joints [-7.71, -25.41, 97.578, 143.544, 84.545, 19.845, -475]
  MoveL 6807 to (-50.81, -35.19, -196.25) mm, rotated rx 105.8 ry 33.04 rz 34.05 deg; joints [-7.701, -25.549, 97.715, 143.553, 84.543, 19.843, -475]
  MoveL 6808 to (-49.25, -36.61, -195.89) mm, rotated rx 105.8 ry 33.04 rz 34.05 deg; joints [-7.689, -25.691, 97.856, 143.565, 84.54, 19.841, -475]
  MoveL 6809 to (-47.64, -38.03, -195.75) mm, rotated rx 105.8 ry 33.04 rz 34.05 deg; joints [-7.685, -25.836, 98.001, 143.569, 84.539, 19.84, -475]
  MoveL 6810 to (-46.05, -39.42, -195.65) mm, rotated rx 105.8 ry 33.04 rz 34.05 deg; joints [-7.682, -25.978, 98.144, 143.571, 84.539, 19.839, -475]
  MoveL 6811 to (-44.43, -40.84, -195.51) mm, rotated rx 105.8 ry 33.04 rz 34.05 deg; joints [-7.678, -26.123, 98.288, 143.575, 84.538, 19.838, -475]
  MoveL 6812 to (-42.88, -42.24, -195.22) mm, rotated rx 105.8 ry 33.04 rz 34.05 deg; joints [-7.668, -26.264, 98.427, 143.585, 84.534, 19.837, -475]
  MoveL 6813 to (-41.21, -43.64, -194.88) mm, rotated rx 105.8 ry 33.04 rz 34.05 deg; joints [-7.656, -26.412, 98.578, 143.596, 84.534, 19.832, -475]
  MoveL 6814 to (-39.6, -45.03, -194.7) mm, rotated rx 105.8 ry 33.04 rz 34.05 deg; joints [-7.65, -26.555, 98.721, 143.602, 84.534, 19.831, -475]
  MoveL 6815 to (-37.97, -46.42, -194.59) mm, rotated rx 105.8 ry 33.04 rz 34.05 deg; joints [-7.648, -26.7, 98.865, 143.605, 84.533, 19.83, -475]
  MoveL 6816 to (-36.36, -47.81, -194.52) mm, rotated rx 105.8 ry 33.04 rz 34.05 deg; joints [-7.646, -26.843, 99.007, 143.606, 84.531, 19.831, -475]
  MoveL 6817 to (-34.73, -49.19, -194.29) mm, rotated rx 105.8 ry 33.04 rz 34.05 deg; joints [-7.639, -26.988, 99.153, 143.614, 84.53, 19.829, -475]
  MoveL 6818 to (-33.11, -50.57, -194.16) mm, rotated rx 105.8 ry 33.04 rz 34.05 deg; joints [-7.635, -27.131, 99.295, 143.617, 84.529, 19.828, -475]
  MoveL 6819 to (-31.48, -51.97, -194.08) mm, rotated rx 105.8 ry 33.04 rz 34.05 deg; joints [-7.633, -27.275, 99.438, 143.619, 84.527, 19.829, -475]
  MoveL 6820 to (-29.85, -53.32, -193.85) mm, rotated rx 105.8 ry 33.04 rz 34.05 deg; joints [-7.625, -27.419, 99.582, 143.626, 84.526, 19.827, -475]
  MoveL 6821 to (-28.19, -54.69, -193.62) mm, rotated rx 105.8 ry 33.04 rz 34.05 deg; joints [-7.618, -27.564, 99.728, 143.634, 84.526, 19.824, -475]
  MoveL 6822 to (-26.52, -56.09, -193.47) mm, rotated rx 105.8 ry 33.04 rz 34.05 deg; joints [-7.613, -27.711, 99.874, 143.638, 84.524, 19.824, -475]
  MoveL 6823 to (-25.06, -57.27, -193.34) mm, rotated rx 105.8 ry 33.04 rz 34.05 deg; joints [-7.61, -27.838, 100.001, 143.642, 84.524, 19.822, -475]
  MoveL 6824 to (-23.75, -58.26, -193.13) mm, rotated rx 105.8 ry 33.04 rz 34.05 deg; joints [-7.603, -27.949, 100.117, 143.649, 84.527, 19.818, -475]
  MoveL 6825 to (-22.55, -59.06, -192.81) mm, rotated rx 105.8 ry 33.04 rz 34.05 deg; joints [-7.592, -28.046, 100.224, 143.66, 84.533, 19.809, -475]
  MoveL 6826 to (-23.51, -57.94, -191.85) mm, rotated rx 105.8 ry 33.04 rz 34.05 deg; joints [-7.554, -27.949, 100.149, 143.698, 84.544, 19.787, -475]
  MoveL 6827 to (-23.13, -58.26, -191.85) mm, rotated rx 105.8 ry 33.04 rz 34.05 deg; joints [-7.555, -27.982, 100.182, 143.697, 84.543, 19.787, -475]
  MoveL 6828 to (-22.78, -58.62, -191.85) mm, rotated rx 105.8 ry 33.04 rz 34.05 deg; joints [-7.555, -28.016, 100.211, 143.697, 84.54, 19.79, -475]
  MoveL 6829 to (-22.49, -59.06, -191.82) mm, rotated rx 105.8 ry 33.04 rz 34.05 deg; joints [-7.554, -28.05, 100.235, 143.698, 84.531, 19.796, -475]
  MoveL 6830 to (-22.23, -59.56, -191.78) mm, rotated rx 105.8 ry 33.04 rz 34.05 deg; joints [-7.552, -28.085, 100.254, 143.698, 84.519, 19.804, -475]
  MoveL 6831 to (-21.99, -60.12, -191.73) mm, rotated rx 105.8 ry 33.04 rz 34.05 deg; joints [-7.55, -28.121, 100.271, 143.7, 84.502, 19.816, -475]
  MoveL 6832 to (-21.81, -60.67, -191.69) mm, rotated rx 105.8 ry 33.04 rz 34.05 deg; joints [-7.548, -28.154, 100.282, 143.7, 84.485, 19.828, -475]
  MoveL 6833 to (-21.65, -61.21, -191.67) mm, rotated rx 105.8 ry 33.04 rz 34.05 deg; joints [-7.547, -28.185, 100.292, 143.7, 84.467, 19.841, -475]
  MoveL 6834 to (-21.51, -61.72, -191.67) mm, rotated rx 105.8 ry 33.04 rz 34.05 deg; joints [-7.546, -28.214, 100.299, 143.699, 84.449, 19.853, -475]
  MoveL 6835 to (-21.37, -62.23, -191.67) mm, rotated rx 105.8 ry 33.04 rz 34.05 deg; joints [-7.546, -28.243, 100.307, 143.698, 84.432, 19.866, -475]
  MoveL 6836 to (-21.18, -62.78, -191.62) mm, rotated rx 105.8 ry 33.04 rz 34.05 deg; joints [-7.544, -28.277, 100.319, 143.699, 84.414, 19.878, -475]
  MoveL 6837 to (-20.95, -63.4, -191.54) mm, rotated rx 105.8 ry 33.04 rz 34.05 deg; joints [-7.54, -28.315, 100.335, 143.701, 84.395, 19.891, -475]
  MoveL 6838 to (-20.78, -63.89, -191.49) mm, rotated rx 105.8 ry 33.04 rz 34.05 deg; joints [-7.538, -28.345, 100.345, 143.702, 84.38, 19.902, -475]
  MoveL 6839 to (-20.66, -64.29, -191.46) mm, rotated rx 105.8 ry 33.04 rz 34.05 deg; joints [-7.537, -28.368, 100.353, 143.702, 84.366, 19.911, -475]
  MoveL 6840 to (-20.52, -64.76, -191.45) mm, rotated rx 105.8 ry 33.04 rz 34.05 deg; joints [-7.536, -28.395, 100.36, 143.702, 84.351, 19.922, -475]
  MoveL 6841 to (-20.38, -65.26, -191.45) mm, rotated rx 105.8 ry 33.04 rz 34.05 deg; joints [-7.536, -28.424, 100.368, 143.701, 84.334, 19.934, -475]
  MoveL 6842 to (-20.24, -65.75, -191.43) mm, rotated rx 105.8 ry 33.04 rz 34.05 deg; joints [-7.535, -28.452, 100.376, 143.701, 84.317, 19.946, -475]
  MoveL 6843 to (-20.09, -66.22, -191.41) mm, rotated rx 105.8 ry 33.04 rz 34.05 deg; joints [-7.533, -28.48, 100.385, 143.701, 84.302, 19.957, -475]
  MoveL 6844 to (-19.95, -66.72, -191.4) mm, rotated rx 105.8 ry 33.04 rz 34.05 deg; joints [-7.533, -28.508, 100.393, 143.701, 84.285, 19.969, -475]
  MoveL 6845 to (-19.26, -69.25, -191.39) mm, rotated rx 105.8 ry 33.04 rz 34.05 deg; joints [-7.531, -28.651, 100.429, 143.696, 84.199, 20.032, -475]
  MoveL 6846 to (-18.94, -70.67, -191.48) mm, rotated rx 105.8 ry 33.04 rz 34.05 deg; joints [-7.533, -28.728, 100.442, 143.69, 84.148, 20.07, -475]
  MoveL 6847 to (-18.82, -71.86, -191.73) mm, rotated rx 105.8 ry 33.04 rz 34.05 deg; joints [-7.541, -28.784, 100.439, 143.678, 84.101, 20.108, -475]
  MoveL 6848 to (-18.89, -72.83, -192.14) mm, rotated rx 105.8 ry 33.04 rz 34.05 deg; joints [-7.556, -28.821, 100.418, 143.66, 84.058, 20.146, -475]
  MoveL 6849 to (-19.16, -73.57, -192.73) mm, rotated rx 105.8 ry 33.04 rz 34.05 deg; joints [-7.577, -28.837, 100.381, 143.637, 84.019, 20.183, -475]
  MoveL 6850 to (-19.63, -74.08, -193.48) mm, rotated rx 105.8 ry 33.04 rz 34.05 deg; joints [-7.605, -28.833, 100.327, 143.607, 83.984, 20.22, -475]
  MoveL 6851 to (-20.29, -74.37, -194.39) mm, rotated rx 105.8 ry 33.04 rz 34.05 deg; joints [-7.638, -28.809, 100.256, 143.571, 83.953, 20.257, -475]
  MoveL 6852 to (-22.2, -74.26, -196.72) mm, rotated rx 105.8 ry 33.04 rz 34.05 deg; joints [-7.724, -28.701, 100.064, 143.482, 83.901, 20.329, -475]
  MoveL 6853 to (-24.3, -73.39, -199.07) mm, rotated rx 105.8 ry 33.04 rz 34.05 deg; joints [-7.811, -28.55, 99.862, 143.394, 83.877, 20.382, -475]
  MoveL 6854 to (-25.99, -71.87, -200.77) mm, rotated rx 105.8 ry 33.04 rz 34.05 deg; joints [-7.875, -28.396, 99.71, 143.332, 83.891, 20.397, -475]
  MoveL 6855 to (-26.69, -70.88, -201.39) mm, rotated rx 105.8 ry 33.04 rz 34.05 deg; joints [-7.898, -28.317, 99.652, 143.31, 83.913, 20.391, -475]
  MoveL 6856 to (-27.28, -69.72, -201.84) mm, rotated rx 105.8 ry 33.04 rz 34.05 deg; joints [-7.916, -28.237, 99.607, 143.295, 83.944, 20.374, -475]
  MoveL 6857 to (-28.14, -66.94, -202.27) mm, rotated rx 105.8 ry 33.04 rz 34.05 deg; joints [-7.934, -28.074, 99.554, 143.285, 84.035, 20.313, -475]
  MoveL 6858 to (-28.36, -65.95, -202.31) mm, rotated rx 105.8 ry 33.04 rz 34.05 deg; joints [-7.936, -28.021, 99.545, 143.285, 84.071, 20.287, -475]
  MoveL 6859 to (-28.72, -63.36, -202.31) mm, rotated rx 105.8 ry 33.04 rz 34.05 deg; joints [-7.939, -27.893, 99.54, 143.29, 84.17, 20.214, -475]
  MoveL 6860 to (-28.9, -62.37, -202.37) mm, rotated rx 105.8 ry 33.04 rz 34.05 deg; joints [-7.942, -27.842, 99.533, 143.29, 84.206, 20.188, -475]
  MoveL 6861 to (-29.04, -61.33, -202.37) mm, rotated rx 105.8 ry 33.04 rz 34.05 deg; joints [-7.943, -27.79, 99.531, 143.292, 84.246, 20.159, -475]
  MoveL 6862 to (-29.12, -60.85, -202.38) mm, rotated rx 105.8 ry 33.04 rz 34.05 deg; joints [-7.944, -27.766, 99.529, 143.292, 84.264, 20.146, -475]
  MoveL 6863 to (-29.19, -60.43, -202.4) mm, rotated rx 105.8 ry 33.04 rz 34.05 deg; joints [-7.945, -27.744, 99.526, 143.292, 84.279, 20.135, -475]
  MoveL 6864 to (-29.27, -59.97, -202.41) mm, rotated rx 105.8 ry 33.04 rz 34.05 deg; joints [-7.946, -27.721, 99.524, 143.293, 84.296, 20.122, -475]
  MoveL 6865 to (-29.63, -57.38, -202.42) mm, rotated rx 105.8 ry 33.04 rz 34.05 deg; joints [-7.949, -27.592, 99.517, 143.297, 84.394, 20.05, -475]
  MoveL 6866 to (-29.72, -56.89, -202.44) mm, rotated rx 105.8 ry 33.04 rz 34.05 deg; joints [-7.95, -27.567, 99.514, 143.297, 84.412, 20.036, -475]
  MoveL 6867 to (-29.82, -56.44, -202.47) mm, rotated rx 105.8 ry 33.04 rz 34.05 deg; joints [-7.952, -27.542, 99.509, 143.297, 84.428, 20.025, -475]
  MoveL 6868 to (-29.95, -56.02, -202.51) mm, rotated rx 105.8 ry 33.04 rz 34.05 deg; joints [-7.954, -27.518, 99.501, 143.296, 84.442, 20.016, -475]
  MoveL 6869 to (-30.11, -55.62, -202.55) mm, rotated rx 105.8 ry 33.04 rz 34.05 deg; joints [-7.955, -27.492, 99.489, 143.295, 84.453, 20.008, -475]
  MoveL 6870 to (-30.33, -55.24, -202.56) mm, rotated rx 105.8 ry 33.04 rz 34.05 deg; joints [-7.956, -27.465, 99.472, 143.295, 84.462, 20.002, -475]
  MoveL 6871 to (-30.59, -54.88, -202.57) mm, rotated rx 105.8 ry 33.04 rz 34.05 deg; joints [-7.956, -27.436, 99.451, 143.296, 84.468, 19.997, -475]
  MoveL 6872 to (-30.26, -55.56, -203.31) mm, rotated rx 105.8 ry 33.04 rz 34.05 deg; joints [-7.984, -27.481, 99.471, 143.267, 84.453, 20.019, -475]
  MoveL 6873 to (-31.39, -54.67, -203.86) mm, rotated rx 105.8 ry 33.04 rz 34.05 deg; joints [-8.004, -27.384, 99.369, 143.247, 84.453, 20.027, -475]
  MoveL 6874 to (-32.55, -53.64, -204.28) mm, rotated rx 105.8 ry 33.04 rz 34.05 deg; joints [-8.019, -27.278, 99.266, 143.232, 84.458, 20.029, -475]
  MoveL 6875 to (-33.82, -52.4, -204.59) mm, rotated rx 105.8 ry 33.04 rz 34.05 deg; joints [-8.03, -27.159, 99.156, 143.222, 84.467, 20.027, -475]
  MoveL 6876 to (-35.2, -50.93, -204.78) mm, rotated rx 105.8 ry 33.04 rz 34.05 deg; joints [-8.036, -27.024, 99.037, 143.217, 84.481, 20.018, -475]
  MoveL 6877 to (-36.63, -49.39, -204.97) mm, rotated rx 105.8 ry 33.04 rz 34.05 deg; joints [-8.043, -26.884, 98.913, 143.212, 84.496, 20.01, -475]
  MoveL 6878 to (-38.06, -47.81, -205.09) mm, rotated rx 105.8 ry 33.04 rz 34.05 deg; joints [-8.046, -26.741, 98.79, 143.209, 84.512, 19.999, -475]
  MoveL 6879 to (-39.5, -46.24, -205.32) mm, rotated rx 105.8 ry 33.04 rz 34.05 deg; joints [-8.054, -26.599, 98.665, 143.203, 84.527, 19.991, -475]
  MoveL 6880 to (-40.93, -44.65, -205.43) mm, rotated rx 105.8 ry 33.04 rz 34.05 deg; joints [-8.058, -26.456, 98.541, 143.2, 84.543, 19.981, -475]
  MoveL 6881 to (-42.36, -43.07, -205.55) mm, rotated rx 105.8 ry 33.04 rz 34.05 deg; joints [-8.061, -26.314, 98.417, 143.198, 84.558, 19.97, -475]
  MoveL 6882 to (-43.79, -41.48, -205.66) mm, rotated rx 105.8 ry 33.04 rz 34.05 deg; joints [-8.065, -26.172, 98.293, 143.195, 84.573, 19.96, -475]
  MoveL 6883 to (-45.22, -39.9, -205.9) mm, rotated rx 105.8 ry 33.04 rz 34.05 deg; joints [-8.073, -26.029, 98.168, 143.188, 84.588, 19.952, -475]
  MoveL 6884 to (-46.64, -38.31, -206.02) mm, rotated rx 105.8 ry 33.04 rz 34.05 deg; joints [-8.077, -25.887, 98.043, 143.186, 84.603, 19.942, -475]
  MoveL 6885 to (-48.05, -36.82, -206.12) mm, rotated rx 105.8 ry 33.04 rz 34.05 deg; joints [-8.08, -25.75, 97.919, 143.184, 84.614, 19.935, -475]
  MoveL 6886 to (-49.52, -35.43, -206.33) mm, rotated rx 105.8 ry 33.04 rz 34.05 deg; joints [-8.086, -25.614, 97.787, 143.177, 84.619, 19.934, -475]
  MoveL 6887 to (-51.17, -33.55, -206.47) mm, rotated rx 105.8 ry 33.04 rz 34.05 deg; joints [-8.091, -25.447, 97.642, 143.174, 84.637, 19.923, -475]
  MoveL 6888 to (-52.68, -31.63, -206.55) mm, rotated rx 105.8 ry 33.04 rz 34.05 deg; joints [-8.093, -25.286, 97.51, 143.173, 84.661, 19.905, -475]
  MoveL 6889 to (-54.14, -29.87, -206.58) mm, rotated rx 105.8 ry 33.04 rz 34.05 deg; joints [-8.094, -25.135, 97.381, 143.174, 84.679, 19.892, -475]
  MoveL 6890 to (-55.5, -28.33, -206.63) mm, rotated rx 105.8 ry 33.04 rz 34.05 deg; joints [-8.095, -24.998, 97.261, 143.174, 84.692, 19.882, -475]
  MoveL 6891 to (-56.8, -26.86, -206.75) mm, rotated rx 105.8 ry 33.04 rz 34.05 deg; joints [-8.098, -24.867, 97.145, 143.171, 84.705, 19.874, -475]
  MoveL 6892 to (-58.15, -25.35, -206.81) mm, rotated rx 105.8 ry 33.04 rz 34.05 deg; joints [-8.1, -24.732, 97.024, 143.171, 84.717, 19.866, -475]
  MoveL 6893 to (-59.55, -23.75, -206.88) mm, rotated rx 105.8 ry 33.04 rz 34.05 deg; joints [-8.102, -24.59, 96.898, 143.17, 84.73, 19.857, -475]
  MoveL 6894 to (-60.85, -22.25, -207.06) mm, rotated rx 105.8 ry 33.04 rz 34.05 deg; joints [-8.108, -24.458, 96.781, 143.164, 84.743, 19.849, -475]
  MoveL 6895 to (-62.08, -20.79, -207.38) mm, rotated rx 105.8 ry 33.04 rz 34.05 deg; joints [-8.12, -24.331, 96.67, 143.154, 84.758, 19.843, -475]
  MoveL 6896 to (-62.23, -19.94, -208.42) mm, rotated rx 105.8 ry 33.04 rz 34.05 deg; joints [-8.16, -24.285, 96.656, 143.117, 84.79, 19.833, -475]
  MoveL 6897 to (-62.02, -20.09, -208.94) mm, rotated rx 105.8 ry 33.04 rz 34.05 deg; joints [-8.179, -24.302, 96.672, 143.098, 84.794, 19.838, -475]
  MoveL 6898 to (-62, -20.08, -209.26) mm, rotated rx 105.8 ry 33.04 rz 34.05 deg; joints [-8.192, -24.302, 96.673, 143.085, 84.796, 19.841, -475]
  MoveL 6899 to (-62.15, -19.93, -209.42) mm, rotated rx 105.8 ry 33.04 rz 34.05 deg; joints [-8.198, -24.287, 96.658, 143.08, 84.797, 19.843, -475]
  MoveL 6900 to (-62.5, -19.69, -209.46) mm, rotated rx 105.8 ry 33.04 rz 34.05 deg; joints [-8.199, -24.259, 96.625, 143.078, 84.793, 19.846, -475]
  MoveL 6901 to (-62.96, -19.45, -209.48) mm, rotated rx 105.8 ry 33.04 rz 34.05 deg; joints [-8.199, -24.225, 96.581, 143.078, 84.786, 19.851, -475]
  MoveL 6902 to (-63.52, -19.24, -209.49) mm, rotated rx 105.8 ry 33.04 rz 34.05 deg; joints [-8.198, -24.186, 96.527, 143.078, 84.774, 19.86, -475]
  MoveL 6903 to (-64.12, -19.05, -209.5) mm, rotated rx 105.8 ry 33.04 rz 34.05 deg; joints [-8.198, -24.147, 96.47, 143.077, 84.759, 19.871, -475]
  MoveL 6904 to (-67.67, -18.14, -209.5) mm, rotated rx 105.8 ry 33.04 rz 34.05 deg; joints [-8.192, -23.922, 96.125, 143.076, 84.661, 19.943, -475]
  MoveL 6905 to (-68.09, -18.01, -209.53) mm, rotated rx 105.8 ry 33.04 rz 34.05 deg; joints [-8.192, -23.895, 96.083, 143.075, 84.65, 19.951, -475]
  MoveL 6906 to (-68.56, -17.89, -209.54) mm, rotated rx 105.8 ry 33.04 rz 34.05 deg; joints [-8.191, -23.865, 96.037, 143.075, 84.638, 19.96, -475]
  MoveL 6907 to (-69.07, -17.75, -209.54) mm, rotated rx 105.8 ry 33.04 rz 34.05 deg; joints [-8.191, -23.833, 95.988, 143.074, 84.624, 19.971, -475]
  MoveL 6908 to (-69.54, -17.62, -209.56) mm, rotated rx 105.8 ry 33.04 rz 34.05 deg; joints [-8.191, -23.802, 95.942, 143.074, 84.612, 19.98, -475]
  MoveL 6909 to (-69.98, -17.47, -209.6) mm, rotated rx 105.8 ry 33.04 rz 34.05 deg; joints [-8.191, -23.773, 95.899, 143.072, 84.601, 19.988, -475]
  MoveL 6910 to (-70.39, -17.33, -209.66) mm, rotated rx 105.8 ry 33.04 rz 34.05 deg; joints [-8.193, -23.745, 95.86, 143.07, 84.591, 19.996, -475]
  MoveL 6911 to (-70.84, -17.19, -209.69) mm, rotated rx 105.8 ry 33.04 rz 34.05 deg; joints [-8.194, -23.716, 95.816, 143.069, 84.58, 20.005, -475]
  MoveL 6912 to (-71.3, -17.05, -209.71) mm, rotated rx 105.8 ry 33.04 rz 34.05 deg; joints [-8.193, -23.685, 95.77, 143.068, 84.568, 20.014, -475]
  MoveL 6913 to (-71.79, -16.92, -209.72) mm, rotated rx 105.8 ry 33.04 rz 34.05 deg; joints [-8.193, -23.654, 95.722, 143.068, 84.554, 20.024, -475]
  MoveL 6914 to (-72.3, -16.79, -209.72) mm, rotated rx 105.8 ry 33.04 rz 34.05 deg; joints [-8.192, -23.622, 95.673, 143.067, 84.54, 20.034, -475]
  MoveL 6915 to (-75.04, -15.79, -210.06) mm, rotated rx 105.8 ry 33.04 rz 34.05 deg; joints [-8.201, -23.435, 95.404, 143.054, 84.477, 20.085, -475]
  MoveL 6916 to (-76.16, -15.13, -210.49) mm, rotated rx 105.8 ry 33.04 rz 34.05 deg; joints [-8.215, -23.347, 95.295, 143.039, 84.462, 20.102, -475]
  MoveL 6917 to (-77.11, -14.36, -211.1) mm, rotated rx 105.8 ry 33.04 rz 34.05 deg; joints [-8.237, -23.264, 95.201, 143.017, 84.458, 20.114, -475]
  MoveL 6918 to (-78.52, -12.51, -212.83) mm, rotated rx 105.8 ry 33.04 rz 34.05 deg; joints [-8.302, -23.108, 95.064, 142.955, 84.484, 20.119, -475]
  MoveL 6919 to (-79.26, -10.22, -215.25) mm, rotated rx 105.8 ry 33.04 rz 34.05 deg; joints [-8.394, -22.969, 94.991, 142.869, 84.555, 20.101, -475]
  MoveL 6920 to (-79.24, -8.19, -217.68) mm, rotated rx 105.8 ry 33.04 rz 34.05 deg; joints [-8.488, -22.879, 94.992, 142.783, 84.645, 20.07, -475]
  MoveL 6921 to (-78.92, -7.51, -218.63) mm, rotated rx 105.8 ry 33.04 rz 34.05 deg; joints [-8.525, -22.865, 95.023, 142.749, 84.687, 20.052, -475]
  MoveL 6922 to (-78.39, -7.07, -219.41) mm, rotated rx 105.8 ry 33.04 rz 34.05 deg; joints [-8.556, -22.873, 95.074, 142.721, 84.728, 20.033, -475]
  MoveL 6923 to (-78.04, -6.93, -219.73) mm, rotated rx 105.8 ry 33.04 rz 34.05 deg; joints [-8.569, -22.885, 95.108, 142.709, 84.747, 20.023, -475]
  MoveL 6924 to (-77.65, -6.85, -220.01) mm, rotated rx 105.8 ry 33.04 rz 34.05 deg; joints [-8.581, -22.902, 95.146, 142.699, 84.767, 20.012, -475]
  MoveL 6925 to (-76.7, -6.86, -220.45) mm, rotated rx 105.8 ry 33.04 rz 34.05 deg; joints [-8.599, -22.951, 95.239, 142.684, 84.804, 19.991, -475]
  MoveL 6926 to (-75.54, -7.1, -220.71) mm, rotated rx 105.8 ry 33.04 rz 34.05 deg; joints [-8.611, -23.022, 95.352, 142.674, 84.84, 19.968, -475]
  MoveL 6927 to (-74.16, -7.57, -220.79) mm, rotated rx 105.8 ry 33.04 rz 34.05 deg; joints [-8.617, -23.114, 95.485, 142.671, 84.874, 19.944, -475]
  MoveL 6928 to (-73.68, -7.77, -220.79) mm, rotated rx 105.8 ry 33.04 rz 34.05 deg; joints [-8.618, -23.147, 95.532, 142.671, 84.885, 19.936, -475]
  MoveL 6929 to (-73.26, -7.95, -220.76) mm, rotated rx 105.8 ry 33.04 rz 34.05 deg; joints [-8.618, -23.177, 95.573, 142.672, 84.894, 19.929, -475]
  MoveL 6930 to (-72.88, -8.14, -220.72) mm, rotated rx 105.8 ry 33.04 rz 34.05 deg; joints [-8.617, -23.205, 95.61, 142.673, 84.901, 19.923, -475]
  MoveL 6931 to (-72.5, -8.34, -220.66) mm, rotated rx 105.8 ry 33.04 rz 34.05 deg; joints [-8.615, -23.234, 95.647, 142.675, 84.907, 19.918, -475]
  MoveL 6932 to (-72.09, -8.53, -220.62) mm, rotated rx 105.8 ry 33.04 rz 34.05 deg; joints [-8.614, -23.263, 95.686, 142.677, 84.915, 19.912, -475]
  MoveL 6933 to (-71.62, -8.73, -220.6) mm, rotated rx 105.8 ry 33.04 rz 34.05 deg; joints [-8.614, -23.296, 95.732, 142.677, 84.925, 19.904, -475]
  MoveL 6934 to (-71.14, -8.92, -220.6) mm, rotated rx 105.8 ry 33.04 rz 34.05 deg; joints [-8.615, -23.33, 95.779, 142.677, 84.936, 19.896, -475]
  MoveL 6935 to (-70.67, -9.11, -220.6) mm, rotated rx 105.8 ry 33.04 rz 34.05 deg; joints [-8.616, -23.362, 95.824, 142.677, 84.946, 19.888, -475]
  MoveL 6936 to (-70.24, -9.3, -220.57) mm, rotated rx 105.8 ry 33.04 rz 34.05 deg; joints [-8.616, -23.393, 95.866, 142.678, 84.955, 19.881, -475]
  MoveL 6937 to (-69.86, -9.48, -220.52) mm, rotated rx 105.8 ry 33.04 rz 34.05 deg; joints [-8.614, -23.421, 95.904, 142.68, 84.962, 19.875, -475]
  MoveL 6938 to (-69.48, -9.66, -220.46) mm, rotated rx 105.8 ry 33.04 rz 34.05 deg; joints [-8.613, -23.449, 95.94, 142.682, 84.969, 19.869, -475]
  MoveL 6939 to (-69.06, -9.87, -220.4) mm, rotated rx 105.8 ry 33.04 rz 34.05 deg; joints [-8.611, -23.479, 95.981, 142.684, 84.977, 19.863, -475]
  MoveL 6940 to (-68.49, -10.12, -220.37) mm, rotated rx 105.8 ry 33.04 rz 34.05 deg; joints [-8.611, -23.52, 96.035, 142.685, 84.988, 19.854, -475]
  MoveL 6941 to (-67.77, -10.44, -220.35) mm, rotated rx 105.8 ry 33.04 rz 34.05 deg; joints [-8.611, -23.571, 96.105, 142.685, 85.003, 19.843, -475]
  MoveL 6942 to (-66.31, -11.02, -220.35) mm, rotated rx 105.8 ry 33.04 rz 34.05 deg; joints [-8.614, -23.672, 96.246, 142.685, 85.035, 19.819, -475]
  MoveL 6943 to (-65.54, -11.33, -220.32) mm, rotated rx 105.8 ry 33.04 rz 34.05 deg; joints [-8.614, -23.726, 96.32, 142.686, 85.051, 19.807, -475]
  MoveL 6944 to (-64.96, -11.58, -220.3) mm, rotated rx 105.8 ry 33.04 rz 34.05 deg; joints [-8.615, -23.766, 96.376, 142.686, 85.063, 19.798, -475]
  MoveL 6945 to (-64.53, -11.8, -220.3) mm, rotated rx 105.8 ry 33.04 rz 34.05 deg; joints [-8.615, -23.798, 96.417, 142.686, 85.071, 19.793, -475]
  MoveL 6946 to (-64.18, -12.03, -220.28) mm, rotated rx 105.8 ry 33.04 rz 34.05 deg; joints [-8.615, -23.826, 96.451, 142.687, 85.075, 19.789, -475]
  MoveL 6947 to (-64.03, -12.18, -220.17) mm, rotated rx 105.8 ry 33.04 rz 34.05 deg; joints [-8.611, -23.841, 96.465, 142.691, 85.074, 19.788, -475]
  MoveL 6948 to (-64.1, -12.18, -219.95) mm, rotated rx 105.8 ry 33.04 rz 34.05 deg; joints [-8.602, -23.837, 96.459, 142.699, 85.071, 19.788, -475]
  MoveL 6949 to (-64.4, -12.02, -219.6) mm, rotated rx 105.8 ry 33.04 rz 34.05 deg; joints [-8.589, -23.816, 96.433, 142.712, 85.065, 19.787, -475]
  MoveL 6950 to (-64.46, -12.8, -218.9) mm, rotated rx 105.8 ry 33.04 rz 34.05 deg; joints [-8.561, -23.847, 96.426, 142.737, 85.029, 19.804, -475]
  MoveL 6951 to (-63.35, -14.48, -218.75) mm, rotated rx 105.8 ry 33.04 rz 34.05 deg; joints [-8.555, -23.977, 96.525, 142.741, 85.003, 19.822, -475]
  MoveL 6952 to (-62.32, -16.11, -218.46) mm, rotated rx 105.8 ry 33.04 rz 34.05 deg; joints [-8.545, -24.101, 96.616, 142.749, 84.975, 19.839, -475]
  MoveL 6953 to (-61.27, -17.72, -218.19) mm, rotated rx 105.8 ry 33.04 rz 34.05 deg; joints [-8.534, -24.226, 96.71, 142.758, 84.949, 19.855, -475]
  MoveL 6954 to (-60.21, -19.34, -217.92) mm, rotated rx 105.8 ry 33.04 rz 34.05 deg; joints [-8.524, -24.351, 96.804, 142.766, 84.922, 19.872, -475]
  MoveL 6955 to (-59.09, -21.03, -217.7) mm, rotated rx 105.8 ry 33.04 rz 34.05 deg; joints [-8.516, -24.482, 96.902, 142.772, 84.894, 19.89, -475]
  MoveL 6956 to (-57.98, -22.84, -217.56) mm, rotated rx 105.8 ry 33.04 rz 34.05 deg; joints [-8.511, -24.618, 96.998, 142.775, 84.862, 19.912, -475]
  MoveL 6957 to (-56.74, -25.05, -217.45) mm, rotated rx 105.8 ry 33.04 rz 34.05 deg; joints [-8.507, -24.777, 97.103, 142.776, 84.818, 19.945, -475]
  MoveL 6958 to (-55.22, -27.02, -217.38) mm, rotated rx 105.8 ry 33.04 rz 34.05 deg; joints [-8.504, -24.941, 97.236, 142.777, 84.793, 19.963, -475]
  MoveL 6959 to (-53.94, -28.7, -217.26) mm, rotated rx 105.8 ry 33.04 rz 34.05 deg; joints [-8.501, -25.08, 97.349, 142.779, 84.772, 19.978, -475]
  MoveL 6960 to (-52.83, -30.23, -217.09) mm, rotated rx 105.8 ry 33.04 rz 34.05 deg; joints [-8.494, -25.204, 97.446, 142.783, 84.749, 19.992, -475]
  MoveL 6961 to (-51.66, -31.91, -216.96) mm, rotated rx 105.8 ry 33.04 rz 34.05 deg; joints [-8.49, -25.336, 97.547, 142.786, 84.723, 20.011, -475]
  MoveL 6962 to (-50.48, -33.62, -216.83) mm, rotated rx 105.8 ry 33.04 rz 34.05 deg; joints [-8.485, -25.472, 97.648, 142.789, 84.695, 20.03, -475]
  MoveL 6963 to (-49.24, -35.41, -216.76) mm, rotated rx 105.8 ry 33.04 rz 34.05 deg; joints [-8.483, -25.612, 97.753, 142.789, 84.666, 20.051, -475]
  MoveL 6964 to (-48.02, -37.16, -216.53) mm, rotated rx 105.8 ry 33.04 rz 34.05 deg; joints [-8.475, -25.751, 97.858, 142.795, 84.638, 20.07, -475]
  MoveL 6965 to (-46.8, -38.92, -216.42) mm, rotated rx 105.8 ry 33.04 rz 34.05 deg; joints [-8.471, -25.89, 97.961, 142.797, 84.609, 20.09, -475]
  MoveL 6966 to (-45.57, -40.66, -216.2) mm, rotated rx 105.8 ry 33.04 rz 34.05 deg; joints [-8.463, -26.028, 98.066, 142.803, 84.58, 20.109, -475]
  MoveL 6967 to (-44.35, -42.41, -216.09) mm, rotated rx 105.8 ry 33.04 rz 34.05 deg; joints [-8.459, -26.167, 98.169, 142.805, 84.551, 20.129, -475]
  MoveL 6968 to (-43.11, -44.15, -215.87) mm, rotated rx 105.8 ry 33.04 rz 34.05 deg; joints [-8.451, -26.306, 98.275, 142.81, 84.523, 20.148, -475]
  MoveL 6969 to (-41.88, -45.89, -215.76) mm, rotated rx 105.8 ry 33.04 rz 34.05 deg; joints [-8.447, -26.445, 98.377, 142.812, 84.494, 20.169, -475]
  MoveL 6970 to (-40.65, -47.64, -215.65) mm, rotated rx 105.8 ry 33.04 rz 34.05 deg; joints [-8.443, -26.583, 98.48, 142.813, 84.464, 20.19, -475]
  MoveL 6971 to (-39.5, -49.17, -215.42) mm, rotated rx 105.8 ry 33.04 rz 34.05 deg; joints [-8.435, -26.709, 98.578, 142.82, 84.44, 20.205, -475]
  MoveL 6972 to (-38.37, -50.61, -215.12) mm, rotated rx 105.8 ry 33.04 rz 34.05 deg; joints [-8.424, -26.829, 98.674, 142.829, 84.419, 20.216, -475]
  MoveL 6973 to (-37.22, -51.99, -214.73) mm, rotated rx 105.8 ry 33.04 rz 34.05 deg; joints [-8.41, -26.949, 98.774, 142.842, 84.401, 20.225, -475]
  MoveL 6974 to (-37.78, -50.69, -213.81) mm, rotated rx 105.8 ry 33.04 rz 34.05 deg; joints [-8.375, -26.866, 98.738, 142.878, 84.432, 20.187, -475]
  MoveL 6975 to (-37.58, -51, -213.75) mm, rotated rx 105.8 ry 33.04 rz 34.05 deg; joints [-8.373, -26.889, 98.755, 142.88, 84.426, 20.191, -475]
  MoveL 6976 to (-37.41, -51.32, -213.69) mm, rotated rx 105.8 ry 33.04 rz 34.05 deg; joints [-8.371, -26.912, 98.769, 142.882, 84.419, 20.196, -475]
  MoveL 6977 to (-37.28, -51.72, -213.66) mm, rotated rx 105.8 ry 33.04 rz 34.05 deg; joints [-8.369, -26.936, 98.777, 142.882, 84.406, 20.205, -475]
  MoveL 6978 to (-37.2, -52.16, -213.63) mm, rotated rx 105.8 ry 33.04 rz 34.05 deg; joints [-8.368, -26.959, 98.781, 142.883, 84.391, 20.216, -475]
  MoveL 6979 to (-37.16, -52.66, -213.63) mm, rotated rx 105.8 ry 33.04 rz 34.05 deg; joints [-8.367, -26.982, 98.779, 142.882, 84.371, 20.231, -475]
  MoveL 6980 to (-37.14, -53.18, -213.62) mm, rotated rx 105.8 ry 33.04 rz 34.05 deg; joints [-8.366, -27.005, 98.776, 142.881, 84.349, 20.247, -475]
  MoveL 6981 to (-37.13, -54.23, -213.62) mm, rotated rx 105.8 ry 33.04 rz 34.05 deg; joints [-8.365, -27.05, 98.766, 142.879, 84.305, 20.28, -475]
  MoveL 6982 to (-37.11, -54.72, -213.6) mm, rotated rx 105.8 ry 33.04 rz 34.05 deg; joints [-8.364, -27.072, 98.763, 142.879, 84.285, 20.294, -475]
  MoveL 6983 to (-37.07, -55.18, -213.56) mm, rotated rx 105.8 ry 33.04 rz 34.05 deg; joints [-8.361, -27.093, 98.762, 142.88, 84.267, 20.308, -475]
  MoveL 6984 to (-37.01, -55.7, -213.48) mm, rotated rx 105.8 ry 33.04 rz 34.05 deg; joints [-8.358, -27.119, 98.763, 142.882, 84.247, 20.322, -475]
  MoveL 6985 to (-36.96, -56.28, -213.41) mm, rotated rx 105.8 ry 33.04 rz 34.05 deg; joints [-8.354, -27.146, 98.762, 142.883, 84.224, 20.338, -475]
  MoveL 6986 to (-36.93, -56.86, -213.38) mm, rotated rx 105.8 ry 33.04 rz 34.05 deg; joints [-8.352, -27.171, 98.758, 142.883, 84.2, 20.355, -475]
  MoveL 6987 to (-36.92, -57.4, -213.37) mm, rotated rx 105.8 ry 33.04 rz 34.05 deg; joints [-8.351, -27.195, 98.754, 142.883, 84.178, 20.371, -475]
  MoveL 6988 to (-36.91, -57.93, -213.36) mm, rotated rx 105.8 ry 33.04 rz 34.05 deg; joints [-8.351, -27.218, 98.749, 142.882, 84.155, 20.388, -475]
  MoveL 6989 to (-36.9, -58.98, -213.36) mm, rotated rx 105.8 ry 33.04 rz 34.05 deg; joints [-8.349, -27.262, 98.739, 142.88, 84.111, 20.421, -475]
  MoveL 6990 to (-36.85, -60.01, -213.34) mm, rotated rx 105.8 ry 33.04 rz 34.05 deg; joints [-8.347, -27.308, 98.732, 142.879, 84.07, 20.452, -475]
  MoveL 6991 to (-36.82, -62.63, -213.34) mm, rotated rx 105.8 ry 33.04 rz 34.05 deg; joints [-8.343, -27.419, 98.706, 142.874, 83.96, 20.534, -475]
  MoveL 6992 to (-36.87, -64.07, -213.43) mm, rotated rx 105.8 ry 33.04 rz 34.05 deg; joints [-8.345, -27.477, 98.685, 142.867, 83.897, 20.583, -475]
  MoveL 6993 to (-37.05, -65.24, -213.69) mm, rotated rx 105.8 ry 33.04 rz 34.05 deg; joints [-8.353, -27.515, 98.652, 142.855, 83.842, 20.628, -475]
  MoveL 6994 to (-37.38, -66.12, -214.13) mm, rotated rx 105.8 ry 33.04 rz 34.05 deg; joints [-8.367, -27.534, 98.608, 142.836, 83.794, 20.67, -475]
  MoveL 6995 to (-37.6, -66.46, -214.41) mm, rotated rx 105.8 ry 33.04 rz 34.05 deg; joints [-8.377, -27.536, 98.581, 142.825, 83.773, 20.69, -475]
  MoveL 6996 to (-37.84, -66.72, -214.74) mm, rotated rx 105.8 ry 33.04 rz 34.05 deg; joints [-8.389, -27.533, 98.552, 142.812, 83.755, 20.709, -475]
  MoveL 6997 to (-38.45, -67.04, -215.53) mm, rotated rx 105.8 ry 33.04 rz 34.05 deg; joints [-8.417, -27.513, 98.486, 142.781, 83.723, 20.745, -475]
  MoveL 6998 to (-39.19, -67.08, -216.5) mm, rotated rx 105.8 ry 33.04 rz 34.05 deg; joints [-8.452, -27.474, 98.408, 142.745, 83.699, 20.777, -475]
  MoveL 6999 to (-41.08, -66.3, -218.95) mm, rotated rx 105.8 ry 33.04 rz 34.05 deg; joints [-8.542, -27.337, 98.218, 142.654, 83.675, 20.833, -475]
  MoveL 7000 to (-42.94, -64.74, -221.41) mm, rotated rx 105.8 ry 33.04 rz 34.05 deg; joints [-8.632, -27.169, 98.04, 142.565, 83.685, 20.863, -475]
  MoveL 7001 to (-44.16, -62.72, -223.16) mm, rotated rx 105.8 ry 33.04 rz 34.05 deg; joints [-8.699, -27.017, 97.932, 142.503, 83.733, 20.854, -475]
  MoveL 7002 to (-44.54, -61.54, -223.78) mm, rotated rx 105.8 ry 33.04 rz 34.05 deg; joints [-8.723, -26.947, 97.904, 142.483, 83.771, 20.834, -475]
  MoveL 7003 to (-44.76, -60.25, -224.22) mm, rotated rx 105.8 ry 33.04 rz 34.05 deg; joints [-8.741, -26.881, 97.895, 142.469, 83.82, 20.804, -475]
  MoveL 7004 to (-44.72, -57.32, -224.57) mm, rotated rx 105.8 ry 33.04 rz 34.05 deg; joints [-8.758, -26.761, 97.928, 142.462, 83.945, 20.714, -475]
  MoveL 7005 to (-44.43, -54.71, -224.56) mm, rotated rx 105.8 ry 33.04 rz 34.05 deg; joints [-8.763, -26.667, 97.984, 142.467, 84.065, 20.624, -475]
  MoveL 7006 to (-44.36, -54.19, -224.55) mm, rotated rx 105.8 ry 33.04 rz 34.05 deg; joints [-8.763, -26.649, 97.996, 142.469, 84.089, 20.605, -475]
  MoveL 7007 to (-44.28, -53.65, -224.52) mm, rotated rx 105.8 ry 33.04 rz 34.05 deg; joints [-8.763, -26.631, 98.01, 142.471, 84.114, 20.586, -475]
  MoveL 7008 to (-44.22, -53.16, -224.51) mm, rotated rx 105.8 ry 33.04 rz 34.05 deg; joints [-8.764, -26.613, 98.021, 142.472, 84.137, 20.568, -475]
  MoveL 7009 to (-44.18, -52.72, -224.53) mm, rotated rx 105.8 ry 33.04 rz 34.05 deg; joints [-8.765, -26.597, 98.03, 142.472, 84.157, 20.553, -475]
  MoveL 7010 to (-44.14, -52.23, -224.56) mm, rotated rx 105.8 ry 33.04 rz 34.05 deg; joints [-8.767, -26.578, 98.038, 142.472, 84.179, 20.537, -475]
  MoveL 7011 to (-44.12, -51.65, -224.63) mm, rotated rx 105.8 ry 33.04 rz 34.05 deg; joints [-8.77, -26.555, 98.046, 142.471, 84.204, 20.519, -475]
  MoveL 7012 to (-44.11, -51.07, -224.71) mm, rotated rx 105.8 ry 33.04 rz 34.05 deg; joints [-8.774, -26.531, 98.052, 142.469, 84.229, 20.502, -475]
  MoveL 7013 to (-44.08, -50.5, -224.75) mm, rotated rx 105.8 ry 33.04 rz 34.05 deg; joints [-8.777, -26.509, 98.061, 142.468, 84.254, 20.484, -475]
  MoveL 7014 to (-44.03, -49.97, -224.78) mm, rotated rx 105.8 ry 33.04 rz 34.05 deg; joints [-8.779, -26.489, 98.07, 142.468, 84.277, 20.466, -475]
  MoveL 7015 to (-43.98, -49.46, -224.79) mm, rotated rx 105.8 ry 33.04 rz 34.05 deg; joints [-8.78, -26.47, 98.081, 142.469, 84.301, 20.448, -475]
  MoveL 7016 to (-43.92, -48.94, -224.79) mm, rotated rx 105.8 ry 33.04 rz 34.05 deg; joints [-8.781, -26.451, 98.091, 142.47, 84.325, 20.43, -475]
  MoveL 7017 to (-43.88, -48.37, -224.82) mm, rotated rx 105.8 ry 33.04 rz 34.05 deg; joints [-8.783, -26.429, 98.101, 142.469, 84.35, 20.412, -475]
  MoveL 7018 to (-43.87, -47.82, -224.87) mm, rotated rx 105.8 ry 33.04 rz 34.05 deg; joints [-8.786, -26.407, 98.108, 142.468, 84.374, 20.395, -475]
  MoveL 7019 to (-43.87, -47.26, -224.94) mm, rotated rx 105.8 ry 33.04 rz 34.05 deg; joints [-8.789, -26.383, 98.112, 142.467, 84.397, 20.378, -475]
  MoveL 7020 to (-43.92, -46.76, -225) mm, rotated rx 105.8 ry 33.04 rz 34.05 deg; joints [-8.792, -26.359, 98.112, 142.465, 84.416, 20.364, -475]
  MoveL 7021 to (-44.02, -46.31, -225.03) mm, rotated rx 105.8 ry 33.04 rz 34.05 deg; joints [-8.794, -26.335, 98.107, 142.465, 84.432, 20.353, -475]
  MoveL 7022 to (-44.16, -45.93, -225.04) mm, rotated rx 105.8 ry 33.04 rz 34.05 deg; joints [-8.794, -26.311, 98.097, 142.465, 84.442, 20.345, -475]
  MoveL 7023 to (-44.32, -45.58, -225.04) mm, rotated rx 105.8 ry 33.04 rz 34.05 deg; joints [-8.794, -26.288, 98.084, 142.466, 84.451, 20.338, -475]
  MoveL 7024 to (-43.93, -46.81, -225.92) mm, rotated rx 105.8 ry 33.04 rz 34.05 deg; joints [-8.827, -26.359, 98.105, 142.431, 84.417, 20.377, -475]
  MoveL 7025 to (-44.77, -45.44, -226.2) mm, rotated rx 105.8 ry 33.04 rz 34.05 deg; joints [-8.837, -26.257, 98.035, 142.423, 84.444, 20.36, -475]
  MoveL 7026 to (-45.67, -43.88, -226.39) mm, rotated rx 105.8 ry 33.04 rz 34.05 deg; joints [-8.845, -26.143, 97.961, 142.418, 84.478, 20.337, -475]
  MoveL 7027 to (-46.65, -42.08, -226.52) mm, rotated rx 105.8 ry 33.04 rz 34.05 deg; joints [-8.85, -26.015, 97.882, 142.416, 84.517, 20.309, -475]
  MoveL 7028 to (-47.7, -40.09, -226.61) mm, rotated rx 105.8 ry 33.04 rz 34.05 deg; joints [-8.854, -25.875, 97.797, 142.415, 84.562, 20.276, -475]
  MoveL 7029 to (-48.71, -38.21, -226.76) mm, rotated rx 105.8 ry 33.04 rz 34.05 deg; joints [-8.86, -25.742, 97.715, 142.412, 84.603, 20.246, -475]
  MoveL 7030 to (-49.74, -36.33, -226.97) mm, rotated rx 105.8 ry 33.04 rz 34.05 deg; joints [-8.868, -25.609, 97.631, 142.407, 84.644, 20.218, -475]
  MoveL 7031 to (-50.69, -34.54, -227.1) mm, rotated rx 105.8 ry 33.04 rz 34.05 deg; joints [-8.873, -25.482, 97.553, 142.405, 84.683, 20.19, -475]
  MoveL 7032 to (-51.59, -32.92, -227.36) mm, rotated rx 105.8 ry 33.04 rz 34.05 deg; joints [-8.883, -25.366, 97.478, 142.397, 84.718, 20.167, -475]
  MoveL 7033 to (-52.56, -31.1, -227.58) mm, rotated rx 105.8 ry 33.04 rz 34.05 deg; joints [-8.891, -25.237, 97.397, 142.392, 84.757, 20.14, -475]
  MoveL 7034 to (-53.53, -29.26, -227.72) mm, rotated rx 105.8 ry 33.04 rz 34.05 deg; joints [-8.897, -25.108, 97.316, 142.389, 84.797, 20.111, -475]
  MoveL 7035 to (-54.52, -27.37, -227.82) mm, rotated rx 105.8 ry 33.04 rz 34.05 deg; joints [-8.901, -24.975, 97.234, 142.388, 84.838, 20.081, -475]
  MoveL 7036 to (-55.51, -25.49, -228.05) mm, rotated rx 105.8 ry 33.04 rz 34.05 deg; joints [-8.91, -24.843, 97.151, 142.382, 84.879, 20.053, -475]
  MoveL 7037 to (-56.49, -23.58, -228.31) mm, rotated rx 105.8 ry 33.04 rz 34.05 deg; joints [-8.921, -24.709, 97.069, 142.375, 84.921, 20.024, -475]
  MoveL 7038 to (-57.47, -21.69, -228.4) mm, rotated rx 105.8 ry 33.04 rz 34.05 deg; joints [-8.924, -24.578, 96.987, 142.374, 84.961, 19.994, -475]
  MoveL 7039 to (-58.47, -19.76, -228.44) mm, rotated rx 105.8 ry 33.04 rz 34.05 deg; joints [-8.926, -24.442, 96.903, 142.375, 85.002, 19.963, -475]
  MoveL 7040 to (-59.43, -17.88, -228.55) mm, rotated rx 105.8 ry 33.04 rz 34.05 deg; joints [-8.931, -24.311, 96.822, 142.373, 85.042, 19.934, -475]
  MoveL 7041 to (-60.39, -15.99, -228.75) mm, rotated rx 105.8 ry 33.04 rz 34.05 deg; joints [-8.939, -24.18, 96.74, 142.368, 85.083, 19.905, -475]
  MoveL 7042 to (-61.32, -14.13, -229.08) mm, rotated rx 105.8 ry 33.04 rz 34.05 deg; joints [-8.952, -24.051, 96.66, 142.357, 85.124, 19.879, -475]
  MoveL 7043 to (-62.27, -12.2, -229.34) mm, rotated rx 105.8 ry 33.04 rz 34.05 deg; joints [-8.962, -23.918, 96.578, 142.35, 85.167, 19.85, -475]
  MoveL 7044 to (-63.21, -10.28, -229.54) mm, rotated rx 105.8 ry 33.04 rz 34.05 deg; joints [-8.97, -23.786, 96.498, 142.345, 85.209, 19.82, -475]
  MoveL 7045 to (-64.15, -8.32, -229.78) mm, rotated rx 105.8 ry 33.04 rz 34.05 deg; joints [-8.98, -23.652, 96.416, 142.338, 85.252, 19.79, -475]
  MoveL 7046 to (-65.11, -6.4, -229.92) mm, rotated rx 105.8 ry 33.04 rz 34.05 deg; joints [-8.986, -23.519, 96.333, 142.335, 85.293, 19.761, -475]
  MoveL 7047 to (-66.08, -4.51, -229.94) mm, rotated rx 105.8 ry 33.04 rz 34.05 deg; joints [-8.987, -23.387, 96.249, 142.336, 85.331, 19.732, -475]
  MoveL 7048 to (-65.99, -3.89, -230.61) mm, rotated rx 105.8 ry 33.04 rz 34.05 deg; joints [-9.013, -23.363, 96.257, 142.312, 85.361, 19.718, -475]
  MoveL 7049 to (-65.77, -4.13, -230.94) mm, rotated rx 105.8 ry 33.04 rz 34.05 deg; joints [-9.026, -23.385, 96.275, 142.3, 85.361, 19.723, -475]
  MoveL 7050 to (-65.73, -4.16, -231.15) mm, rotated rx 105.8 ry 33.04 rz 34.05 deg; joints [-9.034, -23.387, 96.277, 142.292, 85.361, 19.726, -475]
  MoveL 7051 to (-65.88, -3.99, -231.25) mm, rotated rx 105.8 ry 33.04 rz 34.05 deg; joints [-9.037, -23.373, 96.264, 142.288, 85.363, 19.726, -475]
  MoveL 7052 to (-66.2, -3.72, -231.27) mm, rotated rx 105.8 ry 33.04 rz 34.05 deg; joints [-9.038, -23.344, 96.233, 142.288, 85.362, 19.727, -475]
  MoveC 7053 to (-67.05, -3.17, -231.27) mm, rotated rx 105.8 ry 33.04 rz 34.05 deg; joints [-9.036, -23.276, 96.152, 142.289, 85.351, 19.735, -475] to (-67.94, -2.68, -231.27) mm, rotated rx 105.8 ry 33.04 rz 34.05 deg; joints [-9.035, -23.209, 96.066, 142.289, 85.336, 19.746, -475]
  MoveL 7054 to (-67.94, -2.68, -231.27) mm, rotated rx 105.8 ry 33.04 rz 34.05 deg; joints [-9.035, -23.209, 96.066, 142.289, 85.336, 19.746, -475]
  MoveL 7055 to (-68.42, -2.41, -231.3) mm, rotated rx 105.8 ry 33.04 rz 34.05 deg; joints [-9.035, -23.172, 96.021, 142.289, 85.329, 19.751, -475]
  MoveL 7056 to (-68.87, -2.12, -231.35) mm, rotated rx 105.8 ry 33.04 rz 34.05 deg; joints [-9.036, -23.136, 95.977, 142.287, 85.323, 19.756, -475]
  MoveL 7057 to (-69.36, -1.81, -231.41) mm, rotated rx 105.8 ry 33.04 rz 34.05 deg; joints [-9.038, -23.097, 95.93, 142.285, 85.317, 19.762, -475]
  MoveL 7058 to (-69.87, -1.5, -231.46) mm, rotated rx 105.8 ry 33.04 rz 34.05 deg; joints [-9.039, -23.057, 95.881, 142.284, 85.31, 19.767, -475]
  MoveL 7059 to (-70.92, -0.9, -231.48) mm, rotated rx 105.8 ry 33.04 rz 34.05 deg; joints [-9.038, -22.976, 95.78, 142.284, 85.293, 19.78, -475]
  MoveL 7060 to (-71.4, -0.61, -231.51) mm, rotated rx 105.8 ry 33.04 rz 34.05 deg; joints [-9.038, -22.939, 95.734, 142.283, 85.287, 19.785, -475]
  MoveL 7061 to (-71.79, -0.34, -231.58) mm, rotated rx 105.8 ry 33.04 rz 34.05 deg; joints [-9.04, -22.907, 95.696, 142.28, 85.282, 19.789, -475]
  MoveL 7062 to (-72.14, -0.08, -231.67) mm, rotated rx 105.8 ry 33.04 rz 34.05 deg; joints [-9.043, -22.878, 95.662, 142.277, 85.279, 19.793, -475]
  MoveL 7063 to (-72.5, 0.15, -231.74) mm, rotated rx 105.8 ry 33.04 rz 34.05 deg; joints [-9.045, -22.849, 95.627, 142.275, 85.275, 19.797, -475]
  MoveL 7064 to (-72.88, 0.39, -231.77) mm, rotated rx 105.8 ry 33.04 rz 34.05 deg; joints [-9.046, -22.819, 95.59, 142.274, 85.27, 19.801, -475]
  MoveL 7065 to (-75.18, 1.65, -231.77) mm, rotated rx 105.8 ry 33.04 rz 34.05 deg; joints [-9.042, -22.645, 95.368, 142.276, 85.231, 19.83, -475]
  MoveL 7066 to (-77.59, 3.27, -232.12) mm, rotated rx 105.8 ry 33.04 rz 34.05 deg; joints [-9.051, -22.449, 95.134, 142.265, 85.203, 19.855, -475]
  MoveL 7067 to (-78.51, 4.17, -232.55) mm, rotated rx 105.8 ry 33.04 rz 34.05 deg; joints [-9.066, -22.361, 95.044, 142.25, 85.203, 19.861, -475]
  MoveL 7068 to (-79.24, 5.11, -233.15) mm, rotated rx 105.8 ry 33.04 rz 34.05 deg; joints [-9.088, -22.281, 94.972, 142.229, 85.213, 19.861, -475]
  MoveL 7069 to (-79.79, 6.11, -233.93) mm, rotated rx 105.8 ry 33.04 rz 34.05 deg; joints [-9.118, -22.208, 94.917, 142.201, 85.233, 19.857, -475]
  MoveL 7070 to (-80.14, 7.16, -234.88) mm, rotated rx 105.8 ry 33.04 rz 34.05 deg; joints [-9.154, -22.143, 94.88, 142.167, 85.262, 19.848, -475]
  MoveL 7071 to (-80.29, 9.41, -237.29) mm, rotated rx 105.8 ry 33.04 rz 34.05 deg; joints [-9.248, -22.033, 94.859, 142.08, 85.35, 19.815, -475]
  MoveL 7072 to (-79.77, 11.24, -239.7) mm, rotated rx 105.8 ry 33.04 rz 34.05 deg; joints [-9.343, -21.975, 94.903, 141.992, 85.447, 19.774, -475]
  MoveL 7073 to (-79.29, 11.76, -240.65) mm, rotated rx 105.8 ry 33.04 rz 34.05 deg; joints [-9.381, -21.976, 94.947, 141.958, 85.488, 19.756, -475]
  MoveL 7074 to (-78.67, 12.02, -241.43) mm, rotated rx 105.8 ry 33.04 rz 34.05 deg; joints [-9.412, -21.996, 95.006, 141.929, 85.524, 19.74, -475]
  MoveL 7075 to (-78.3, 12.05, -241.75) mm, rotated rx 105.8 ry 33.04 rz 34.05 deg; joints [-9.425, -22.013, 95.04, 141.917, 85.54, 19.732, -475]
  MoveL 7076 to (-77.89, 12.02, -242.03) mm, rotated rx 105.8 ry 33.04 rz 34.05 deg; joints [-9.437, -22.035, 95.079, 141.906, 85.555, 19.724, -475]
  MoveL 7077 to (-76.97, 11.75, -242.46) mm, rotated rx 105.8 ry 33.04 rz 34.05 deg; joints [-9.455, -22.093, 95.166, 141.89, 85.582, 19.711, -475]
  MoveL 7078 to (-75.9, 11.22, -242.72) mm, rotated rx 105.8 ry 33.04 rz 34.05 deg; joints [-9.467, -22.171, 95.269, 141.879, 85.603, 19.698, -475]
  MoveL 7079 to (-74.68, 10.42, -242.81) mm, rotated rx 105.8 ry 33.04 rz 34.05 deg; joints [-9.473, -22.268, 95.386, 141.875, 85.62, 19.687, -475]
  MoveL 7080 to (-74.26, 10.12, -242.81) mm, rotated rx 105.8 ry 33.04 rz 34.05 deg; joints [-9.473, -22.304, 95.427, 141.875, 85.624, 19.684, -475]
  MoveL 7081 to (-73.91, 9.84, -242.77) mm, rotated rx 105.8 ry 33.04 rz 34.05 deg; joints [-9.473, -22.334, 95.461, 141.875, 85.627, 19.682, -475]
  MoveL 7082 to (-73.59, 9.57, -242.72) mm, rotated rx 105.8 ry 33.04 rz 34.05 deg; joints [-9.471, -22.363, 95.491, 141.877, 85.628, 19.68, -475]
  MoveL 7083 to (-73.28, 9.29, -242.65) mm, rotated rx 105.8 ry 33.04 rz 34.05 deg; joints [-9.469, -22.39, 95.521, 141.879, 85.629, 19.678, -475]
  MoveL 7084 to (-72.94, 9.01, -242.6) mm, rotated rx 105.8 ry 33.04 rz 34.05 deg; joints [-9.468, -22.42, 95.554, 141.881, 85.631, 19.676, -475]
  MoveL 7085 to (-72.54, 8.71, -242.58) mm, rotated rx 105.8 ry 33.04 rz 34.05 deg; joints [-9.468, -22.455, 95.593, 141.881, 85.635, 19.673, -475]
  MoveL 7086 to (-67.88, 5.36, -242.57) mm, rotated rx 105.8 ry 33.04 rz 34.05 deg; joints [-9.475, -22.84, 96.037, 141.877, 85.683, 19.638, -475]
  MoveL 7087 to (-67.27, 4.91, -242.56) mm, rotated rx 105.8 ry 33.04 rz 34.05 deg; joints [-9.476, -22.892, 96.096, 141.876, 85.688, 19.634, -475]
  MoveL 7088 to (-66.76, 4.49, -242.55) mm, rotated rx 105.8 ry 33.04 rz 34.05 deg; joints [-9.476, -22.936, 96.144, 141.876, 85.691, 19.632, -475]
  MoveL 7089 to (-66.38, 4.06, -242.54) mm, rotated rx 105.8 ry 33.04 rz 34.05 deg; joints [-9.476, -22.975, 96.18, 141.876, 85.689, 19.634, -475]
  MoveL 7090 to (-66.07, 3.62, -242.5) mm, rotated rx 105.8 ry 33.04 rz 34.05 deg; joints [-9.475, -23.01, 96.208, 141.877, 85.683, 19.638, -475]
  MoveL 7091 to (-65.94, 3.31, -242.34) mm, rotated rx 105.8 ry 33.04 rz 34.05 deg; joints [-9.468, -23.031, 96.221, 141.883, 85.676, 19.641, -475]
  MoveL 7092 to (-65.96, 3.3, -242.03) mm, rotated rx 105.8 ry 33.04 rz 34.05 deg; joints [-9.457, -23.031, 96.221, 141.894, 85.674, 19.638, -475]
  MoveL 7093 to (-66.15, 3.61, -241.54) mm, rotated rx 105.8 ry 33.04 rz 34.05 deg; joints [-9.438, -23.008, 96.207, 141.913, 85.678, 19.629, -475]
  MoveL 7094 to (-66.54, 3.12, -240.57) mm, rotated rx 105.8 ry 33.04 rz 34.05 deg; joints [-9.4, -23.011, 96.173, 141.949, 85.641, 19.643, -475]
  MoveL 7095 to (-65.93, 1.35, -240.27) mm, rotated rx 105.8 ry 33.04 rz 34.05 deg; joints [-9.387, -23.12, 96.225, 141.958, 85.595, 19.675, -475]
  MoveL 7096 to (-65.28, -0.49, -240.07) mm, rotated rx 105.8 ry 33.04 rz 34.05 deg; joints [-9.378, -23.235, 96.281, 141.964, 85.546, 19.71, -475]
  MoveL 7097 to (-64.55, -2.49, -239.94) mm, rotated rx 105.8 ry 33.04 rz 34.05 deg; joints [-9.372, -23.36, 96.341, 141.967, 85.495, 19.748, -475]
  MoveL 7098 to (-63.05, -6.49, -239.94) mm, rotated rx 105.8 ry 33.04 rz 34.05 deg; joints [-9.37, -23.611, 96.463, 141.962, 85.393, 19.827, -475]
  MoveL 7099 to (-62.36, -8.35, -239.85) mm, rotated rx 105.8 ry 33.04 rz 34.05 deg; joints [-9.365, -23.727, 96.52, 141.964, 85.345, 19.863, -475]
  MoveL 7100 to (-61.61, -10.35, -239.85) mm, rotated rx 105.8 ry 33.04 rz 34.05 deg; joints [-9.364, -23.852, 96.58, 141.962, 85.293, 19.903, -475]
  MoveL 7101 to (-60.95, -12.4, -239.85) mm, rotated rx 105.8 ry 33.04 rz 34.05 deg; joints [-9.363, -23.975, 96.631, 141.959, 85.236, 19.947, -475]
  MoveL 7102 to (-60.21, -14.84, -239.67) mm, rotated rx 105.8 ry 33.04 rz 34.05 deg; joints [-9.354, -24.119, 96.688, 141.963, 85.166, 19.999, -475]
  MoveL 7103 to (-59.31, -16.87, -239.44) mm, rotated rx 105.8 ry 33.04 rz 34.05 deg; joints [-9.345, -24.254, 96.763, 141.969, 85.118, 20.033, -475]
  MoveL 7104 to (-58.46, -18.87, -239.32) mm, rotated rx 105.8 ry 33.04 rz 34.05 deg; joints [-9.339, -24.384, 96.833, 141.972, 85.069, 20.07, -475]
  MoveL 7105 to (-57.71, -20.87, -239.21) mm, rotated rx 105.8 ry 33.04 rz 34.05 deg; joints [-9.334, -24.509, 96.892, 141.973, 85.016, 20.109, -475]
  MoveL 7106 to (-56.95, -22.87, -239) mm, rotated rx 105.8 ry 33.04 rz 34.05 deg; joints [-9.325, -24.634, 96.952, 141.979, 84.963, 20.147, -475]
  MoveL 7107 to (-56.2, -24.86, -238.89) mm, rotated rx 105.8 ry 33.04 rz 34.05 deg; joints [-9.32, -24.759, 97.011, 141.98, 84.91, 20.187, -475]
  MoveL 7108 to (-55.44, -26.86, -238.78) mm, rotated rx 105.8 ry 33.04 rz 34.05 deg; joints [-9.314, -24.884, 97.07, 141.981, 84.857, 20.227, -475]
  MoveL 7109 to (-54.68, -28.85, -238.57) mm, rotated rx 105.8 ry 33.04 rz 34.05 deg; joints [-9.305, -25.01, 97.13, 141.987, 84.804, 20.265, -475]
  MoveL 7110 to (-53.92, -30.84, -238.46) mm, rotated rx 105.8 ry 33.04 rz 34.05 deg; joints [-9.3, -25.135, 97.188, 141.988, 84.75, 20.305, -475]
  MoveL 7111 to (-53.16, -32.83, -238.36) mm, rotated rx 105.8 ry 33.04 rz 34.05 deg; joints [-9.295, -25.259, 97.246, 141.989, 84.697, 20.345, -475]
  MoveL 7112 to (-52.38, -34.82, -238.15) mm, rotated rx 105.8 ry 33.04 rz 34.05 deg; joints [-9.286, -25.385, 97.307, 141.994, 84.644, 20.383, -475]
  MoveL 7113 to (-51.61, -36.81, -238.05) mm, rotated rx 105.8 ry 33.04 rz 34.05 deg; joints [-9.281, -25.51, 97.364, 141.995, 84.59, 20.423, -475]
  MoveL 7114 to (-50.88, -38.51, -237.79) mm, rotated rx 105.8 ry 33.04 rz 34.05 deg; joints [-9.271, -25.621, 97.422, 142.002, 84.546, 20.453, -475]
  MoveL 7115 to (-50.16, -40.02, -237.43) mm, rotated rx 105.8 ry 33.04 rz 34.05 deg; joints [-9.257, -25.723, 97.481, 142.013, 84.509, 20.477, -475]
  MoveL 7116 to (-49.44, -41.36, -236.92) mm, rotated rx 105.8 ry 33.04 rz 34.05 deg; joints [-9.238, -25.818, 97.542, 142.03, 84.479, 20.493, -475]
  MoveL 7117 to (-49.6, -40.24, -236.08) mm, rotated rx 105.8 ry 33.04 rz 34.05 deg; joints [-9.207, -25.764, 97.544, 142.063, 84.517, 20.451, -475]
  MoveL 7118 to (-49.48, -40.55, -236.05) mm, rotated rx 105.8 ry 33.04 rz 34.05 deg; joints [-9.206, -25.783, 97.552, 142.063, 84.508, 20.457, -475]
  MoveL 7119 to (-49.4, -40.86, -236.01) mm, rotated rx 105.8 ry 33.04 rz 34.05 deg; joints [-9.204, -25.801, 97.558, 142.065, 84.498, 20.464, -475]
  MoveL 7120 to (-49.39, -41.23, -235.95) mm, rotated rx 105.8 ry 33.04 rz 34.05 deg; joints [-9.201, -25.817, 97.556, 142.066, 84.483, 20.475, -475]
  MoveL 7121 to (-49.43, -41.65, -235.92) mm, rotated rx 105.8 ry 33.04 rz 34.05 deg; joints [-9.199, -25.833, 97.549, 142.067, 84.464, 20.489, -475]
  MoveL 7122 to (-49.51, -42.12, -235.89) mm, rotated rx 105.8 ry 33.04 rz 34.05 deg; joints [-9.197, -25.849, 97.536, 142.067, 84.442, 20.506, -475]
  MoveL 7123 to (-50.6, -46.71, -235.89) mm, rotated rx 105.8 ry 33.04 rz 34.05 deg; joints [-9.187, -25.985, 97.385, 142.059, 84.214, 20.68, -475]
  MoveL 7124 to (-50.67, -47.11, -235.87) mm, rotated rx 105.8 ry 33.04 rz 34.05 deg; joints [-9.185, -25.997, 97.374, 142.059, 84.195, 20.694, -475]
  MoveL 7125 to (-50.79, -47.61, -235.87) mm, rotated rx 105.8 ry 33.04 rz 34.05 deg; joints [-9.184, -26.012, 97.358, 142.059, 84.169, 20.714, -475]
  MoveL 7126 to (-51, -48.62, -235.83) mm, rotated rx 105.8 ry 33.04 rz 34.05 deg; joints [-9.181, -26.043, 97.327, 142.058, 84.12, 20.751, -475]
  MoveL 7127 to (-51.61, -51.17, -235.83) mm, rotated rx 105.8 ry 33.04 rz 34.05 deg; joints [-9.175, -26.118, 97.242, 142.053, 83.993, 20.848, -475]
  MoveL 7128 to (-51.79, -52.19, -235.81) mm, rotated rx 105.8 ry 33.04 rz 34.05 deg; joints [-9.172, -26.151, 97.214, 142.052, 83.945, 20.885, -475]
  MoveL 7129 to (-52.1, -53.6, -235.87) mm, rotated rx 105.8 ry 33.04 rz 34.05 deg; joints [-9.172, -26.192, 97.168, 142.047, 83.875, 20.939, -475]
  MoveL 7130 to (-52.5, -54.7, -236.13) mm, rotated rx 105.8 ry 33.04 rz 34.05 deg; joints [-9.179, -26.217, 97.116, 142.035, 83.816, 20.988, -475]
  MoveL 7131 to (-52.97, -55.5, -236.57) mm, rotated rx 105.8 ry 33.04 rz 34.05 deg; joints [-9.193, -26.224, 97.058, 142.017, 83.768, 21.032, -475]
  MoveL 7132 to (-53.23, -55.79, -236.86) mm, rotated rx 105.8 ry 33.04 rz 34.05 deg; joints [-9.202, -26.221, 97.026, 142.006, 83.748, 21.052, -475]
  MoveL 7133 to (-53.52, -55.99, -237.19) mm, rotated rx 105.8 ry 33.04 rz 34.05 deg; joints [-9.214, -26.213, 96.994, 141.993, 83.73, 21.071, -475]
  MoveL 7134 to (-54.15, -56.18, -238.01) mm, rotated rx 105.8 ry 33.04 rz 34.05 deg; joints [-9.242, -26.186, 96.924, 141.962, 83.702, 21.105, -475]
  MoveL 7135 to (-54.86, -56.07, -239) mm, rotated rx 105.8 ry 33.04 rz 34.05 deg; joints [-9.278, -26.141, 96.848, 141.925, 83.685, 21.133, -475]
  MoveL 7136 to (-56.51, -54.91, -241.56) mm, rotated rx 105.8 ry 33.04 rz 34.05 deg; joints [-9.371, -26, 96.678, 141.833, 83.682, 21.176, -475]
  MoveL 7137 to (-57.96, -53, -244.13) mm, rotated rx 105.8 ry 33.04 rz 34.05 deg; joints [-9.467, -25.838, 96.536, 141.741, 83.717, 21.188, -475]
  MoveL 7138 to (-58.68, -50.78, -245.96) mm, rotated rx 105.8 ry 33.04 rz 34.05 deg; joints [-9.537, -25.704, 96.473, 141.678, 83.787, 21.162, -475]
  MoveL 7139 to (-58.77, -49.56, -246.6) mm, rotated rx 105.8 ry 33.04 rz 34.05 deg; joints [-9.563, -25.647, 96.472, 141.657, 83.836, 21.134, -475]
  MoveL 7140 to (-58.68, -48.26, -247.06) mm, rotated rx 105.8 ry 33.04 rz 34.05 deg; joints [-9.582, -25.597, 96.49, 141.642, 83.894, 21.096, -475]
  MoveL 7141 to (-57.95, -45.43, -247.42) mm, rotated rx 105.8 ry 33.04 rz 34.05 deg; joints [-9.603, -25.517, 96.587, 141.634, 84.037, 20.991, -475]
  MoveL 7142 to (-56.87, -42.48, -247.42) mm, rotated rx 105.8 ry 33.04 rz 34.05 deg; joints [-9.611, -25.451, 96.722, 141.639, 84.196, 20.868, -475]
  MoveL 7143 to (-56.54, -41.51, -247.44) mm, rotated rx 105.8 ry 33.04 rz 34.05 deg; joints [-9.614, -25.428, 96.763, 141.64, 84.247, 20.828, -475]
  MoveL 7144 to (-56.18, -40.53, -247.44) mm, rotated rx 105.8 ry 33.04 rz 34.05 deg; joints [-9.616, -25.406, 96.808, 141.641, 84.3, 20.787, -475]
  MoveL 7145 to (-56.01, -40.06, -247.44) mm, rotated rx 105.8 ry 33.04 rz 34.05 deg; joints [-9.618, -25.395, 96.829, 141.642, 84.325, 20.768, -475]
  MoveL 7146 to (-55.8, -39.43, -247.47) mm, rotated rx 105.8 ry 33.04 rz 34.05 deg; joints [-9.621, -25.38, 96.856, 141.642, 84.358, 20.742, -475]
  MoveL 7147 to (-55.62, -38.86, -247.53) mm, rotated rx 105.8 ry 33.04 rz 34.05 deg; joints [-9.624, -25.365, 96.878, 141.641, 84.388, 20.72, -475]
  MoveL 7148 to (-55.49, -38.38, -247.6) mm, rotated rx 105.8 ry 33.04 rz 34.05 deg; joints [-9.628, -25.351, 96.895, 141.639, 84.413, 20.702, -475]
  MoveL 7149 to (-55.36, -37.93, -247.65) mm, rotated rx 105.8 ry 33.04 rz 34.05 deg; joints [-9.631, -25.339, 96.911, 141.637, 84.436, 20.685, -475]
  MoveL 7150 to (-55.22, -37.49, -247.69) mm, rotated rx 105.8 ry 33.04 rz 34.05 deg; joints [-9.634, -25.328, 96.929, 141.637, 84.459, 20.668, -475]
  MoveL 7151 to (-54.68, -36.01, -247.69) mm, rotated rx 105.8 ry 33.04 rz 34.05 deg; joints [-9.638, -25.294, 96.995, 141.639, 84.539, 20.606, -475]
  MoveL 7152 to (-54.53, -35.53, -247.7) mm, rotated rx 105.8 ry 33.04 rz 34.05 deg; joints [-9.64, -25.282, 97.015, 141.639, 84.564, 20.587, -475]
  MoveL 7153 to (-54.42, -35.11, -247.73) mm, rotated rx 105.8 ry 33.04 rz 34.05 deg; joints [-9.642, -25.27, 97.029, 141.638, 84.585, 20.571, -475]
  MoveL 7154 to (-54.35, -34.73, -247.77) mm, rotated rx 105.8 ry 33.04 rz 34.05 deg; joints [-9.644, -25.257, 97.039, 141.637, 84.603, 20.557, -475]
  MoveL 7155 to (-54.36, -34.42, -247.84) mm, rotated rx 105.8 ry 33.04 rz 34.05 deg; joints [-9.647, -25.243, 97.04, 141.635, 84.615, 20.549, -475]
  MoveL 7156 to (-54.41, -34.15, -247.91) mm, rotated rx 105.8 ry 33.04 rz 34.05 deg; joints [-9.65, -25.229, 97.037, 141.633, 84.624, 20.543, -475]
  MoveL 7157 to (-54.73, -35.71, -248.71) mm, rotated rx 105.8 ry 33.04 rz 34.05 deg; joints [-9.677, -25.276, 96.985, 141.601, 84.552, 20.611, -475]
  MoveL 7158 to (-55.11, -33.98, -249.12) mm, rotated rx 105.8 ry 33.04 rz 34.05 deg; joints [-9.694, -25.183, 96.96, 141.589, 84.609, 20.573, -475]
  MoveL 7159 to (-55.54, -32.16, -249.38) mm, rotated rx 105.8 ry 33.04 rz 34.05 deg; joints [-9.706, -25.082, 96.931, 141.582, 84.668, 20.531, -475]
  MoveL 7160 to (-56.03, -30.22, -249.56) mm, rotated rx 105.8 ry 33.04 rz 34.05 deg; joints [-9.714, -24.974, 96.899, 141.577, 84.729, 20.485, -475]
  MoveL 7161 to (-56.57, -28.16, -249.76) mm, rotated rx 105.8 ry 33.04 rz 34.05 deg; joints [-9.724, -24.857, 96.862, 141.573, 84.793, 20.438, -475]
  MoveL 7162 to (-57.09, -26.08, -249.85) mm, rotated rx 105.8 ry 33.04 rz 34.05 deg; joints [-9.729, -24.742, 96.827, 141.572, 84.857, 20.389, -475]
  MoveL 7163 to (-57.61, -24.02, -249.95) mm, rotated rx 105.8 ry 33.04 rz 34.05 deg; joints [-9.735, -24.626, 96.792, 141.571, 84.921, 20.34, -475]
  MoveL 7164 to (-58.14, -21.95, -250.15) mm, rotated rx 105.8 ry 33.04 rz 34.05 deg; joints [-9.744, -24.51, 96.755, 141.566, 84.985, 20.293, -475]
  MoveL 7165 to (-58.66, -19.88, -250.25) mm, rotated rx 105.8 ry 33.04 rz 34.05 deg; joints [-9.75, -24.394, 96.719, 141.565, 85.049, 20.244, -475]
  MoveL 7166 to (-59.17, -17.81, -250.35) mm, rotated rx 105.8 ry 33.04 rz 34.05 deg; joints [-9.756, -24.278, 96.684, 141.564, 85.113, 20.196, -475]
  MoveL 7167 to (-59.69, -15.74, -250.55) mm, rotated rx 105.8 ry 33.04 rz 34.05 deg; joints [-9.765, -24.162, 96.647, 141.559, 85.177, 20.148, -475]
  MoveL 7168 to (-60.71, -11.59, -250.75) mm, rotated rx 105.8 ry 33.04 rz 34.05 deg; joints [-9.777, -23.93, 96.575, 141.556, 85.304, 20.051, -475]
  MoveL 7169 to (-61.13, -9.85, -250.96) mm, rotated rx 105.8 ry 33.04 rz 34.05 deg; joints [-9.786, -23.832, 96.543, 141.55, 85.358, 20.012, -475]
  MoveL 7170 to (-61.63, -7.95, -251.03) mm, rotated rx 105.8 ry 33.04 rz 34.05 deg; joints [-9.791, -23.724, 96.506, 141.549, 85.414, 19.969, -475]
  MoveL 7171 to (-62.22, -5.98, -251.04) mm, rotated rx 105.8 ry 33.04 rz 34.05 deg; joints [-9.793, -23.609, 96.462, 141.55, 85.47, 19.925, -475]
  MoveL 7172 to (-62.84, -3.38, -251.15) mm, rotated rx 105.8 ry 33.04 rz 34.05 deg; joints [-9.8, -23.464, 96.416, 141.549, 85.549, 19.865, -475]
  MoveL 7173 to (-63.33, -0.85, -251.24) mm, rotated rx 105.8 ry 33.04 rz 34.05 deg; joints [-9.806, -23.328, 96.383, 141.547, 85.63, 19.802, -475]
  MoveL 7174 to (-63.81, 1.31, -251.34) mm, rotated rx 105.8 ry 33.04 rz 34.05 deg; joints [-9.812, -23.209, 96.348, 141.546, 85.697, 19.751, -475]
  MoveL 7175 to (-64.27, 3.3, -251.51) mm, rotated rx 105.8 ry 33.04 rz 34.05 deg; joints [-9.82, -23.098, 96.312, 141.541, 85.758, 19.706, -475]
  MoveL 7176 to (-64.69, 5.16, -251.79) mm, rotated rx 105.8 ry 33.04 rz 34.05 deg; joints [-9.833, -22.995, 96.279, 141.532, 85.815, 19.665, -475]
  MoveL 7177 to (-65.1, 7.01, -252.08) mm, rotated rx 105.8 ry 33.04 rz 34.05 deg; joints [-9.846, -22.892, 96.247, 141.523, 85.872, 19.624, -475]
  MoveL 7178 to (-65.48, 8.85, -252.37) mm, rotated rx 105.8 ry 33.04 rz 34.05 deg; joints [-9.859, -22.791, 96.217, 141.513, 85.931, 19.583, -475]
  MoveL 7179 to (-65.91, 10.79, -252.53) mm, rotated rx 105.8 ry 33.04 rz 34.05 deg; joints [-9.867, -22.684, 96.183, 141.508, 85.99, 19.539, -475]
  MoveL 7180 to (-65.58, 11.35, -253.15) mm, rotated rx 105.8 ry 33.04 rz 34.05 deg; joints [-9.892, -22.675, 96.214, 141.485, 86.025, 19.52, -475]
  MoveL 7181 to (-65.37, 11.11, -253.46) mm, rotated rx 105.8 ry 33.04 rz 34.05 deg; joints [-9.904, -22.695, 96.23, 141.473, 86.024, 19.525, -475]
  MoveL 7182 to (-65.33, 11.11, -253.65) mm, rotated rx 105.8 ry 33.04 rz 34.05 deg; joints [-9.912, -22.697, 96.233, 141.466, 86.027, 19.526, -475]
  MoveL 7183 to (-65.44, 11.34, -253.75) mm, rotated rx 105.8 ry 33.04 rz 34.05 deg; joints [-9.915, -22.681, 96.223, 141.463, 86.031, 19.523, -475]
  MoveL 7184 to (-65.7, 11.7, -253.77) mm, rotated rx 105.8 ry 33.04 rz 34.05 deg; joints [-9.916, -22.652, 96.198, 141.463, 86.035, 19.52, -475]
  MoveL 7185 to (-66.02, 12.07, -253.77) mm, rotated rx 105.8 ry 33.04 rz 34.05 deg; joints [-9.916, -22.619, 96.168, 141.463, 86.037, 19.519, -475]
  MoveL 7186 to (-66.74, 12.73, -253.8) mm, rotated rx 105.8 ry 33.04 rz 34.05 deg; joints [-9.916, -22.553, 96.1, 141.463, 86.036, 19.52, -475]
  MoveL 7187 to (-67.9, 13.79, -253.8) mm, rotated rx 105.8 ry 33.04 rz 34.05 deg; joints [-9.914, -22.447, 95.99, 141.464, 86.032, 19.522, -475]
  MoveL 7188 to (-68.6, 14.48, -253.82) mm, rotated rx 105.8 ry 33.04 rz 34.05 deg; joints [-9.914, -22.381, 95.924, 141.465, 86.032, 19.522, -475]
  MoveL 7189 to (-69.37, 15.18, -253.82) mm, rotated rx 105.8 ry 33.04 rz 34.05 deg; joints [-9.913, -22.31, 95.851, 141.466, 86.03, 19.523, -475]
  MoveL 7190 to (-69.75, 15.54, -253.84) mm, rotated rx 105.8 ry 33.04 rz 34.05 deg; joints [-9.913, -22.275, 95.815, 141.466, 86.029, 19.524, -475]
  MoveL 7191 to (-70.09, 15.87, -253.86) mm, rotated rx 105.8 ry 33.04 rz 34.05 deg; joints [-9.913, -22.244, 95.783, 141.465, 86.029, 19.524, -475]
  MoveL 7192 to (-70.4, 16.18, -253.91) mm, rotated rx 105.8 ry 33.04 rz 34.05 deg; joints [-9.915, -22.214, 95.753, 141.464, 86.029, 19.525, -475]
  MoveL 7193 to (-70.67, 16.47, -253.97) mm, rotated rx 105.8 ry 33.04 rz 34.05 deg; joints [-9.917, -22.187, 95.726, 141.462, 86.03, 19.525, -475]
  MoveL 7194 to (-70.96, 16.77, -254.03) mm, rotated rx 105.8 ry 33.04 rz 34.05 deg; joints [-9.918, -22.158, 95.698, 141.46, 86.03, 19.525, -475]
  MoveL 7195 to (-71.29, 17.1, -254.06) mm, rotated rx 105.8 ry 33.04 rz 34.05 deg; joints [-9.919, -22.127, 95.667, 141.459, 86.03, 19.525, -475]
  MoveL 7196 to (-71.64, 17.43, -254.08) mm, rotated rx 105.8 ry 33.04 rz 34.05 deg; joints [-9.92, -22.095, 95.634, 141.459, 86.03, 19.526, -475]
  MoveL 7197 to (-71.94, 17.74, -254.13) mm, rotated rx 105.8 ry 33.04 rz 34.05 deg; joints [-9.921, -22.065, 95.605, 141.458, 86.03, 19.526, -475]
  MoveL 7198 to (-72.21, 18.04, -254.19) mm, rotated rx 105.8 ry 33.04 rz 34.05 deg; joints [-9.923, -22.038, 95.579, 141.456, 86.032, 19.525, -475]
  MoveL 7199 to (-72.48, 18.34, -254.24) mm, rotated rx 105.8 ry 33.04 rz 34.05 deg; joints [-9.924, -22.011, 95.552, 141.454, 86.033, 19.525, -475]
  MoveL 7200 to (-72.8, 18.66, -254.27) mm, rotated rx 105.8 ry 33.04 rz 34.05 deg; joints [-9.925, -21.981, 95.522, 141.454, 86.033, 19.525, -475]
  MoveL 7201 to (-73.18, 19.01, -254.27) mm, rotated rx 105.8 ry 33.04 rz 34.05 deg; joints [-9.924, -21.945, 95.485, 141.454, 86.031, 19.526, -475]
  MoveL 7202 to (-75.16, 21.16, -254.63) mm, rotated rx 105.8 ry 33.04 rz 34.05 deg; joints [-9.935, -21.749, 95.295, 141.444, 86.038, 19.525, -475]
  MoveL 7203 to (-75.86, 22.24, -255.07) mm, rotated rx 105.8 ry 33.04 rz 34.05 deg; joints [-9.952, -21.664, 95.225, 141.428, 86.052, 19.52, -475]
  MoveL 7204 to (-76.39, 23.31, -255.69) mm, rotated rx 105.8 ry 33.04 rz 34.05 deg; joints [-9.976, -21.588, 95.172, 141.406, 86.074, 19.511, -475]
  MoveL 7205 to (-76.88, 25.48, -257.48) mm, rotated rx 105.8 ry 33.04 rz 34.05 deg; joints [-10.045, -21.464, 95.116, 141.341, 86.14, 19.483, -475]
  MoveL 7206 to (-76.63, 27.66, -259.97) mm, rotated rx 105.8 ry 33.04 rz 34.05 deg; joints [-10.144, -21.375, 95.128, 141.249, 86.237, 19.441, -475]
  MoveL 7207 to (-75.82, 29.26, -262.46) mm, rotated rx 105.8 ry 33.04 rz 34.05 deg; joints [-10.244, -21.339, 95.193, 141.156, 86.332, 19.4, -475]
  MoveL 7208 to (-75.28, 29.64, -263.44) mm, rotated rx 105.8 ry 33.04 rz 34.05 deg; joints [-10.283, -21.348, 95.239, 141.119, 86.369, 19.385, -475]
  MoveL 7209 to (-74.65, 29.73, -264.24) mm, rotated rx 105.8 ry 33.04 rz 34.05 deg; joints [-10.316, -21.374, 95.296, 141.088, 86.398, 19.373, -475]
  MoveL 7210 to (-74.3, 29.67, -264.58) mm, rotated rx 105.8 ry 33.04 rz 34.05 deg; joints [-10.33, -21.394, 95.327, 141.076, 86.409, 19.368, -475]
  MoveL 7211 to (-73.93, 29.53, -264.87) mm, rotated rx 105.8 ry 33.04 rz 34.05 deg; joints [-10.342, -21.418, 95.362, 141.064, 86.419, 19.365, -475]
  MoveL 7212 to (-73.11, 29.05, -265.31) mm, rotated rx 105.8 ry 33.04 rz 34.05 deg; joints [-10.36, -21.48, 95.437, 141.047, 86.433, 19.36, -475]
  MoveL 7213 to (-72.21, 28.28, -265.58) mm, rotated rx 105.8 ry 33.04 rz 34.05 deg; joints [-10.372, -21.56, 95.522, 141.035, 86.439, 19.359, -475]
  MoveL 7214 to (-71.21, 27.23, -265.67) mm, rotated rx 105.8 ry 33.04 rz 34.05 deg; joints [-10.377, -21.657, 95.617, 141.031, 86.438, 19.362, -475]
  MoveL 7215 to (-69.49, 25.25, -265.67) mm, rotated rx 105.8 ry 33.04 rz 34.05 deg; joints [-10.379, -21.832, 95.78, 141.028, 86.429, 19.37, -475]
  MoveL 7216 to (-69.21, 24.91, -265.64) mm, rotated rx 105.8 ry 33.04 rz 34.05 deg; joints [-10.378, -21.862, 95.807, 141.029, 86.427, 19.371, -475]
  MoveL 7217 to (-68.97, 24.59, -265.59) mm, rotated rx 105.8 ry 33.04 rz 34.05 deg; joints [-10.376, -21.889, 95.83, 141.03, 86.424, 19.373, -475]
  MoveL 7218 to (-68.74, 24.28, -265.52) mm, rotated rx 105.8 ry 33.04 rz 34.05 deg; joints [-10.374, -21.914, 95.852, 141.032, 86.421, 19.375, -475]
  MoveL 7219 to (-68.48, 23.94, -265.47) mm, rotated rx 105.8 ry 33.04 rz 34.05 deg; joints [-10.372, -21.943, 95.877, 141.034, 86.418, 19.377, -475]
  MoveL 7220 to (-68.16, 23.55, -265.43) mm, rotated rx 105.8 ry 33.04 rz 34.05 deg; joints [-10.371, -21.976, 95.907, 141.035, 86.415, 19.379, -475]
  MoveL 7221 to (-67.84, 23.13, -265.37) mm, rotated rx 105.8 ry 33.04 rz 34.05 deg; joints [-10.369, -22.011, 95.938, 141.036, 86.411, 19.381, -475]
  MoveL 7222 to (-67.49, 22.72, -265.36) mm, rotated rx 105.8 ry 33.04 rz 34.05 deg; joints [-10.369, -22.047, 95.971, 141.037, 86.409, 19.383, -475]
  MoveL 7223 to (-67.07, 22.24, -265.37) mm, rotated rx 105.8 ry 33.04 rz 34.05 deg; joints [-10.37, -22.09, 96.011, 141.035, 86.407, 19.385, -475]
  MoveL 7224 to (-66.48, 21.6, -265.44) mm, rotated rx 105.8 ry 33.04 rz 34.05 deg; joints [-10.374, -22.148, 96.066, 141.032, 86.405, 19.387, -475]
  MoveL 7225 to (-66.13, 21.2, -265.44) mm, rotated rx 105.8 ry 33.04 rz 34.05 deg; joints [-10.374, -22.183, 96.099, 141.031, 86.403, 19.389, -475]
  MoveL 7226 to (-65.81, 20.83, -265.43) mm, rotated rx 105.8 ry 33.04 rz 34.05 deg; joints [-10.374, -22.217, 96.129, 141.031, 86.401, 19.391, -475]
  MoveL 7227 to (-65.51, 20.47, -265.41) mm, rotated rx 105.8 ry 33.04 rz 34.05 deg; joints [-10.374, -22.248, 96.158, 141.032, 86.399, 19.393, -475]
  MoveL 7228 to (-65.26, 20.14, -265.36) mm, rotated rx 105.8 ry 33.04 rz 34.05 deg; joints [-10.372, -22.276, 96.182, 141.033, 86.396, 19.395, -475]
  MoveL 7229 to (-65.03, 19.81, -265.3) mm, rotated rx 105.8 ry 33.04 rz 34.05 deg; joints [-10.37, -22.302, 96.203, 141.035, 86.392, 19.397, -475]
  MoveL 7230 to (-64.83, 19.44, -265.25) mm, rotated rx 105.8 ry 33.04 rz 34.05 deg; joints [-10.368, -22.329, 96.222, 141.036, 86.385, 19.402, -475]
  MoveL 7231 to (-64.67, 19.06, -265.19) mm, rotated rx 105.8 ry 33.04 rz 34.05 deg; joints [-10.366, -22.354, 96.237, 141.038, 86.376, 19.408, -475]
  MoveL 7232 to (-64.64, 18.84, -265.03) mm, rotated rx 105.8 ry 33.04 rz 34.05 deg; joints [-10.359, -22.365, 96.24, 141.044, 86.369, 19.412, -475]
